REGION Network 29: T-03.00 Transfer Pump Cmd and Speed
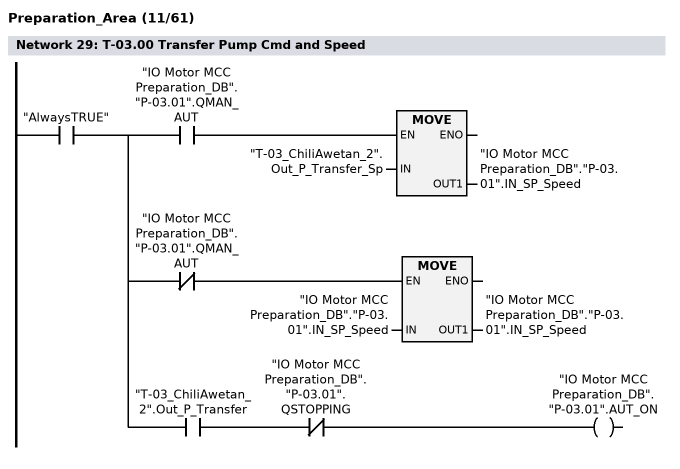
   RUNG wire#powerrail
      Contact( "AlwaysTRUE" )
      wire#w1
      Contact( "IO Motor MCC Preparation_DB"."P-03.01".QMAN_AUT )
      Move(in := "T-03_ChiliAwetan_2".Out_P_Transfer_Sp, out1 => "IO Motor MCC Preparation_DB"."P-03.01".IN_SP_Speed)
   END_RUNG
   RUNG wire#w1
      I_Contact( "IO Motor MCC Preparation_DB"."P-03.01".QMAN_AUT )
      Move(in := "IO Motor MCC Preparation_DB"."P-03.01".IN_SP_Speed, out1 => "IO Motor MCC Preparation_DB"."P-03.01".IN_SP_Speed)
   END_RUNG
   RUNG wire#w1
      Contact( "T-03_ChiliAwetan_2".Out_P_Transfer )
      I_Contact( "IO Motor MCC Preparation_DB"."P-03.01".QSTOPPING )
      Coil( "IO Motor MCC Preparation_DB"."P-03.01".AUT_ON )
   END_RUNG
   // the same network as SCL:
   IF "AlwaysTRUE" AND "IO Motor MCC Preparation_DB"."P-03.01".QMAN_AUT THEN
       "IO Motor MCC Preparation_DB"."P-03.01".IN_SP_Speed := "T-03_ChiliAwetan_2".Out_P_Transfer_Sp;
   END_IF;
   IF "AlwaysTRUE" AND NOT "IO Motor MCC Preparation_DB"."P-03.01".QMAN_AUT THEN
       "IO Motor MCC Preparation_DB"."P-03.01".IN_SP_Speed := "IO Motor MCC Preparation_DB"."P-03.01".IN_SP_Speed;
   END_IF;
   "IO Motor MCC Preparation_DB"."P-03.01".AUT_ON := "AlwaysTRUE" AND "T-03_ChiliAwetan_2".Out_P_Transfer AND NOT "IO Motor MCC Preparation_DB"."P-03.01".QSTOPPING;
END_REGION

REGION Network 30: T-03.00 Feedback Instrument
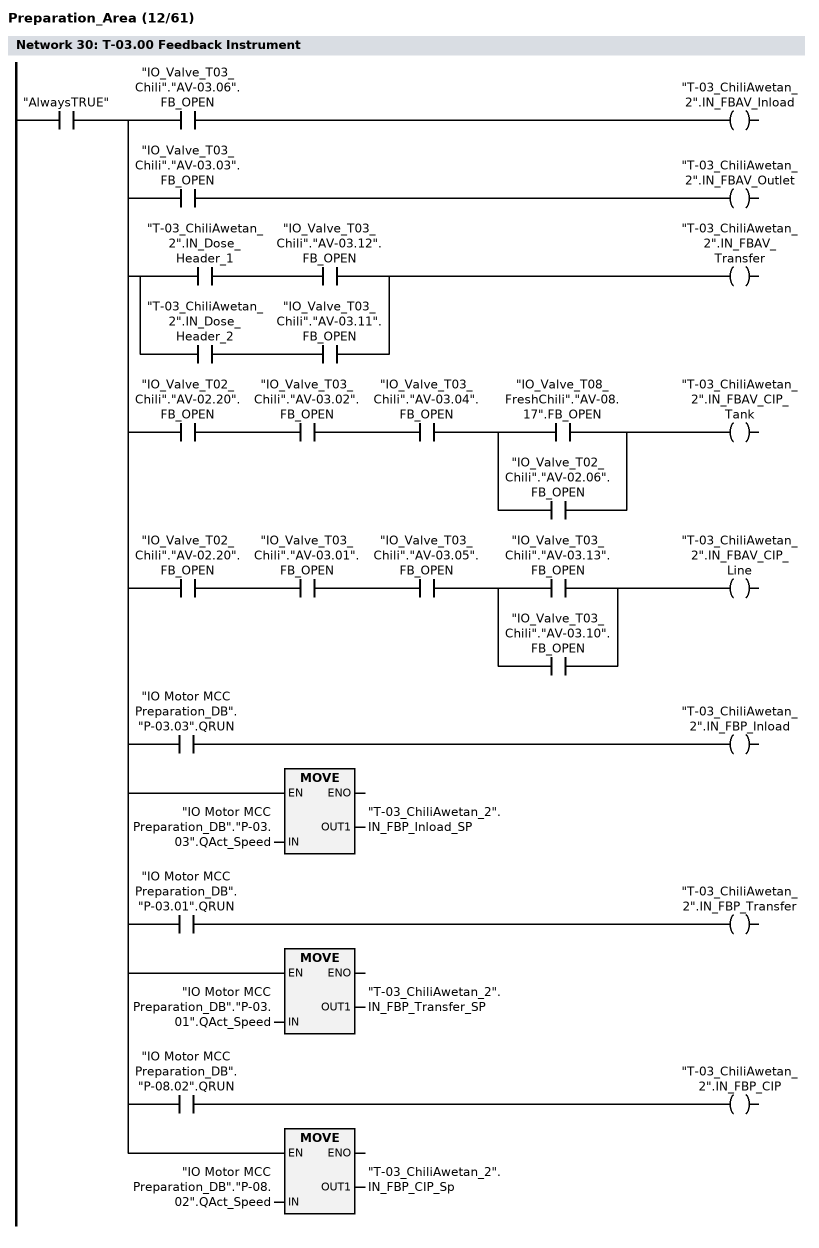
   RUNG wire#powerrail
      Contact( "AlwaysTRUE" )
      wire#w1
      Contact( "IO_Valve_T03_Chili"."AV-03.06".FB_OPEN )
      Coil( "T-03_ChiliAwetan_2".IN_FBAV_Inload )
   END_RUNG
   RUNG wire#w1
      Contact( "IO_Valve_T03_Chili"."AV-03.03".FB_OPEN )
      Coil( "T-03_ChiliAwetan_2".IN_FBAV_Outlet )
   END_RUNG
   RUNG wire#w1
      Contact( "T-03_ChiliAwetan_2".IN_Dose_Header_1 )
      Contact( "IO_Valve_T03_Chili"."AV-03.12".FB_OPEN )
      wire#w2
      Coil( "T-03_ChiliAwetan_2".IN_FBAV_Transfer )
   END_RUNG
   RUNG wire#w1
      Contact( "T-03_ChiliAwetan_2".IN_Dose_Header_2 )
      Contact( "IO_Valve_T03_Chili"."AV-03.11".FB_OPEN )
   END_RUNG wire#w2
   RUNG wire#w1
      Contact( "IO_Valve_T02_Chili"."AV-02.20".FB_OPEN )
      Contact( "IO_Valve_T03_Chili"."AV-03.02".FB_OPEN )
      Contact( "IO_Valve_T03_Chili"."AV-03.04".FB_OPEN )
      wire#w3
      Contact( "IO_Valve_T08_FreshChili"."AV-08.17".FB_OPEN )
      wire#w4
      Coil( "T-03_ChiliAwetan_2".IN_FBAV_CIP_Tank )
   END_RUNG
   RUNG wire#w3
      Contact( "IO_Valve_T02_Chili"."AV-02.06".FB_OPEN )
   END_RUNG wire#w4
   RUNG wire#w1
      Contact( "IO_Valve_T02_Chili"."AV-02.20".FB_OPEN )
      Contact( "IO_Valve_T03_Chili"."AV-03.01".FB_OPEN )
      Contact( "IO_Valve_T03_Chili"."AV-03.05".FB_OPEN )
      wire#w5
      Contact( "IO_Valve_T03_Chili"."AV-03.13".FB_OPEN )
      wire#w6
      Coil( "T-03_ChiliAwetan_2".IN_FBAV_CIP_Line )
   END_RUNG
   RUNG wire#w5
      Contact( "IO_Valve_T03_Chili"."AV-03.10".FB_OPEN )
   END_RUNG wire#w6
   RUNG wire#w1
      Contact( "IO Motor MCC Preparation_DB"."P-03.03".QRUN )
      Coil( "T-03_ChiliAwetan_2".IN_FBP_Inload )
   END_RUNG
   RUNG wire#w1
      Move(in := "IO Motor MCC Preparation_DB"."P-03.03".QAct_Speed, out1 => "T-03_ChiliAwetan_2".IN_FBP_Inload_SP)
   END_RUNG
   RUNG wire#w1
      Contact( "IO Motor MCC Preparation_DB"."P-03.01".QRUN )
      Coil( "T-03_ChiliAwetan_2".IN_FBP_Transfer )
   END_RUNG
   RUNG wire#w1
      Move(in := "IO Motor MCC Preparation_DB"."P-03.01".QAct_Speed, out1 => "T-03_ChiliAwetan_2".IN_FBP_Transfer_SP)
   END_RUNG
   RUNG wire#w1
      Contact( "IO Motor MCC Preparation_DB"."P-08.02".QRUN )
      Coil( "T-03_ChiliAwetan_2".IN_FBP_CIP )
   END_RUNG
   RUNG wire#w1
      Move(in := "IO Motor MCC Preparation_DB"."P-08.02".QAct_Speed, out1 => "T-03_ChiliAwetan_2".IN_FBP_CIP_Sp)
   END_RUNG
   // the same network as SCL:
   "T-03_ChiliAwetan_2".IN_FBAV_Inload := "AlwaysTRUE" AND "IO_Valve_T03_Chili"."AV-03.06".FB_OPEN;
   "T-03_ChiliAwetan_2".IN_FBAV_Outlet := "AlwaysTRUE" AND "IO_Valve_T03_Chili"."AV-03.03".FB_OPEN;
   "T-03_ChiliAwetan_2".IN_FBAV_Transfer := "AlwaysTRUE" AND (("T-03_ChiliAwetan_2".IN_Dose_Header_1 AND "IO_Valve_T03_Chili"."AV-03.12".FB_OPEN) OR ("T-03_ChiliAwetan_2".IN_Dose_Header_2 AND "IO_Valve_T03_Chili"."AV-03.11".FB_OPEN));
   "T-03_ChiliAwetan_2".IN_FBAV_CIP_Tank := "AlwaysTRUE" AND "IO_Valve_T02_Chili"."AV-02.20".FB_OPEN AND "IO_Valve_T03_Chili"."AV-03.02".FB_OPEN AND "IO_Valve_T03_Chili"."AV-03.04".FB_OPEN AND ("IO_Valve_T08_FreshChili"."AV-08.17".FB_OPEN OR "IO_Valve_T02_Chili"."AV-02.06".FB_OPEN);
   "T-03_ChiliAwetan_2".IN_FBAV_CIP_Line := "AlwaysTRUE" AND "IO_Valve_T02_Chili"."AV-02.20".FB_OPEN AND "IO_Valve_T03_Chili"."AV-03.01".FB_OPEN AND "IO_Valve_T03_Chili"."AV-03.05".FB_OPEN AND ("IO_Valve_T03_Chili"."AV-03.13".FB_OPEN OR "IO_Valve_T03_Chili"."AV-03.10".FB_OPEN);
   "T-03_ChiliAwetan_2".IN_FBP_Inload := "AlwaysTRUE" AND "IO Motor MCC Preparation_DB"."P-03.03".QRUN;
   IF "AlwaysTRUE" THEN
       "T-03_ChiliAwetan_2".IN_FBP_Inload_SP := "IO Motor MCC Preparation_DB"."P-03.03".QAct_Speed;
   END_IF;
   "T-03_ChiliAwetan_2".IN_FBP_Transfer := "AlwaysTRUE" AND "IO Motor MCC Preparation_DB"."P-03.01".QRUN;
   IF "AlwaysTRUE" THEN
       "T-03_ChiliAwetan_2".IN_FBP_Transfer_SP := "IO Motor MCC Preparation_DB"."P-03.01".QAct_Speed;
   END_IF;
   "T-03_ChiliAwetan_2".IN_FBP_CIP := "AlwaysTRUE" AND "IO Motor MCC Preparation_DB"."P-08.02".QRUN;
   IF "AlwaysTRUE" THEN
       "T-03_ChiliAwetan_2".IN_FBP_CIP_Sp := "IO Motor MCC Preparation_DB"."P-08.02".QAct_Speed;
   END_IF;
END_REGION

REGION Network 31: T-03.00 Comm to Blend
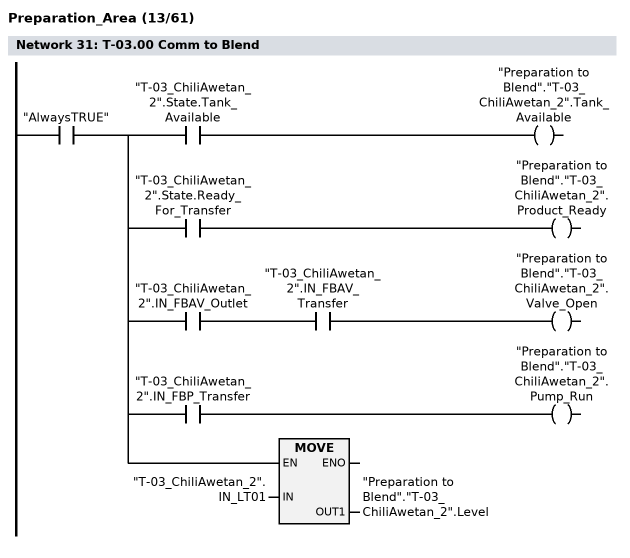
   RUNG wire#powerrail
      Contact( "AlwaysTRUE" )
      wire#w1
      Contact( "T-03_ChiliAwetan_2".State.Tank_Available )
      Coil( "Preparation to Blend"."T-03_ChiliAwetan_2".Tank_Available )
   END_RUNG
   RUNG wire#w1
      Contact( "T-03_ChiliAwetan_2".State.Ready_For_Transfer )
      Coil( "Preparation to Blend"."T-03_ChiliAwetan_2".Product_Ready )
   END_RUNG
   RUNG wire#w1
      Contact( "T-03_ChiliAwetan_2".IN_FBAV_Outlet )
      Contact( "T-03_ChiliAwetan_2".IN_FBAV_Transfer )
      Coil( "Preparation to Blend"."T-03_ChiliAwetan_2".Valve_Open )
   END_RUNG
   RUNG wire#w1
      Contact( "T-03_ChiliAwetan_2".IN_FBP_Transfer )
      Coil( "Preparation to Blend"."T-03_ChiliAwetan_2".Pump_Run )
   END_RUNG
   RUNG wire#w1
      Move(in := "T-03_ChiliAwetan_2".IN_LT01, out1 => "Preparation to Blend"."T-03_ChiliAwetan_2".Level)
   END_RUNG
   // the same network as SCL:
   "Preparation to Blend"."T-03_ChiliAwetan_2".Tank_Available := "AlwaysTRUE" AND "T-03_ChiliAwetan_2".State.Tank_Available;
   "Preparation to Blend"."T-03_ChiliAwetan_2".Product_Ready := "AlwaysTRUE" AND "T-03_ChiliAwetan_2".State.Ready_For_Transfer;
   "Preparation to Blend"."T-03_ChiliAwetan_2".Valve_Open := "AlwaysTRUE" AND "T-03_ChiliAwetan_2".IN_FBAV_Outlet AND "T-03_ChiliAwetan_2".IN_FBAV_Transfer;
   "Preparation to Blend"."T-03_ChiliAwetan_2".Pump_Run := "AlwaysTRUE" AND "T-03_ChiliAwetan_2".IN_FBP_Transfer;
   IF "AlwaysTRUE" THEN
       "Preparation to Blend"."T-03_ChiliAwetan_2".Level := "T-03_ChiliAwetan_2".IN_LT01;
   END_IF;
END_REGION

NETWORK
TITLE = T-04.00 DOSE ON OFF
      O     "Blend to Preparation"."T-20".Raw_Material.ChiliAwetan_3.DoseRun;
      O     "Blend to Preparation"."T-21".Raw_Material.ChiliAwetan_3.DoseRun;
      O     "Blend to Preparation"."T-30".Raw_Material.ChiliAwetan_3.DoseRun;
      O     "Blend to Preparation"."T-31".Raw_Material.ChiliAwetan_3.DoseRun;
      O     "Blend to Preparation"."T-40".Raw_Material.ChiliAwetan_3.DoseRun;
      O     "Blend to Preparation"."T-41".Raw_Material.ChiliAwetan_3.DoseRun;
      =     "T-04_ChiliAwetan_3".IN_Dose_Run;

NETWORK
TITLE = T-04.00 DOSE PAUSE
      O     "Blend to Preparation"."T-20".Raw_Material.ChiliAwetan_3.DoseHeld;
      O     "Blend to Preparation"."T-21".Raw_Material.ChiliAwetan_3.DoseHeld;
      O     "Blend to Preparation"."T-30".Raw_Material.ChiliAwetan_3.DoseHeld;
      O     "Blend to Preparation"."T-31".Raw_Material.ChiliAwetan_3.DoseHeld;
      O     "Blend to Preparation"."T-40".Raw_Material.ChiliAwetan_3.DoseHeld;
      O     "Blend to Preparation"."T-41".Raw_Material.ChiliAwetan_3.DoseHeld;
      =     "T-04_ChiliAwetan_3".IN_Dose_Held;

NETWORK
TITLE = T-04.00 DOSE VALVE CMD
      O(;
      A     "Blend to Preparation"."T-20".Raw_Material.ChiliAwetan_3.DoseRun;
      A     "Blend to Preparation"."T-20".Raw_Material.ChiliAwetan_3.ValveCMD;
      );
      O(;
      A     "Blend to Preparation"."T-21".Raw_Material.ChiliAwetan_3.DoseRun;
      A     "Blend to Preparation"."T-21".Raw_Material.ChiliAwetan_3.ValveCMD;
      );
      O(;
      A     "Blend to Preparation"."T-30".Raw_Material.ChiliAwetan_3.DoseRun;
      A     "Blend to Preparation"."T-30".Raw_Material.ChiliAwetan_3.ValveCMD;
      );
      O(;
      A     "Blend to Preparation"."T-31".Raw_Material.ChiliAwetan_3.DoseRun;
      A     "Blend to Preparation"."T-31".Raw_Material.ChiliAwetan_3.ValveCMD;
      );
      O(;
      A     "Blend to Preparation"."T-40".Raw_Material.ChiliAwetan_3.DoseRun;
      A     "Blend to Preparation"."T-40".Raw_Material.ChiliAwetan_3.ValveCMD;
      );
      O(;
      A     "Blend to Preparation"."T-41".Raw_Material.ChiliAwetan_3.DoseRun;
      A     "Blend to Preparation"."T-41".Raw_Material.ChiliAwetan_3.ValveCMD;
      );
      =     "T-04_ChiliAwetan_3".IN_Dose_Valve_Cmd;



NETWORK
TITLE = T-04.00 DOSE Pump CMD
      O(;
      A     "Blend to Preparation"."T-20".Raw_Material.ChiliAwetan_3.DoseRun;
      A     "Blend to Preparation"."T-20".Raw_Material.ChiliAwetan_3.PumpCMD;
      );
      O(;
      A     "Blend to Preparation"."T-21".Raw_Material.ChiliAwetan_3.DoseRun;
      A     "Blend to Preparation"."T-21".Raw_Material.ChiliAwetan_3.PumpCMD;
      );
      O(;
      A     "Blend to Preparation"."T-30".Raw_Material.ChiliAwetan_3.DoseRun;
      A     "Blend to Preparation"."T-30".Raw_Material.ChiliAwetan_3.PumpCMD;
      );
      O(;
      A     "Blend to Preparation"."T-31".Raw_Material.ChiliAwetan_3.DoseRun;
      A     "Blend to Preparation"."T-31".Raw_Material.ChiliAwetan_3.PumpCMD;
      );
      O(;
      A     "Blend to Preparation"."T-40".Raw_Material.ChiliAwetan_3.DoseRun;
      A     "Blend to Preparation"."T-40".Raw_Material.ChiliAwetan_3.PumpCMD;
      );
      O(;
      A     "Blend to Preparation"."T-41".Raw_Material.ChiliAwetan_3.DoseRun;
      A     "Blend to Preparation"."T-41".Raw_Material.ChiliAwetan_3.PumpCMD;
      );
      =     "T-04_ChiliAwetan_3".IN_Dose_Pump_Cmd;



NETWORK
TITLE = T-04.00 DOSE PUMP SPEED
// Checking
      O     "Blend to Preparation"."T-20".Raw_Material.ChiliAwetan_3.DoseRun;
      JC    SP_04_FROM_20;
      O     "Blend to Preparation"."T-21".Raw_Material.ChiliAwetan_3.DoseRun;
      JC    SP_04_FROM_21;
      O     "Blend to Preparation"."T-30".Raw_Material.ChiliAwetan_3.DoseRun;
      JC    SP_04_FROM_30;
      O     "Blend to Preparation"."T-31".Raw_Material.ChiliAwetan_3.DoseRun;
      JC    SP_04_FROM_31;
      O     "Blend to Preparation"."T-40".Raw_Material.ChiliAwetan_3.DoseRun;
      JC    SP_04_FROM_40;
      O     "Blend to Preparation"."T-41".Raw_Material.ChiliAwetan_3.DoseRun;
      JC    SP_04_FROM_41;
//Jump to end if Blend not Dosing
      JC    SP_04_SELF;
//Load Set Point
SP_04_FROM_20:L     "Blend to Preparation".Recipe."T-20".ChiliAwetan_3.SP_PumpSpeed;
      T     "T-04_ChiliAwetan_3".IN_Dose_Pump_Sp;
      JC    SP_04_SELF;
SP_04_FROM_21:L     "Blend to Preparation".Recipe."T-21".ChiliAwetan_3.SP_PumpSpeed;
      T     "T-04_ChiliAwetan_3".IN_Dose_Pump_Sp;
      JC    SP_04_SELF;
SP_04_FROM_30:L     "Blend to Preparation".Recipe."T-30".ChiliAwetan_3.SP_PumpSpeed;
      T     "T-04_ChiliAwetan_3".IN_Dose_Pump_Sp;
      JC    SP_04_SELF;
SP_04_FROM_31:L     "Blend to Preparation".Recipe."T-31".ChiliAwetan_3.SP_PumpSpeed;
      T     "T-04_ChiliAwetan_3".IN_Dose_Pump_Sp;
      JC    SP_04_SELF;
SP_04_FROM_40:L     "Blend to Preparation".Recipe."T-40".ChiliAwetan_3.SP_PumpSpeed;
      T     "T-04_ChiliAwetan_3".IN_Dose_Pump_Sp;
      JC    SP_04_SELF;
SP_04_FROM_41:L     "Blend to Preparation".Recipe."T-41".ChiliAwetan_3.SP_PumpSpeed;
      T     "T-04_ChiliAwetan_3".IN_Dose_Pump_Sp;
      JC    SP_04_SELF;
// END
SP_04_SELF:L     "T-04_ChiliAwetan_3".IN_Dose_Pump_Sp;
      T     "T-04_ChiliAwetan_3".IN_Dose_Pump_Sp;


NETWORK
TITLE = T-04.00 Header Req
// HEADER 1 Req
      O     "Blend to Preparation"."T-20".Raw_Material.ChiliAwetan_3.Header1_Req;
      O     "Blend to Preparation"."T-21".Raw_Material.ChiliAwetan_3.Header1_Req;
      O     "Blend to Preparation"."T-30".Raw_Material.ChiliAwetan_3.Header1_Req;
      O     "Blend to Preparation"."T-31".Raw_Material.ChiliAwetan_3.Header1_Req;
      O     "Blend to Preparation"."T-40".Raw_Material.ChiliAwetan_3.Header1_Req;
      O     "Blend to Preparation"."T-41".Raw_Material.ChiliAwetan_3.Header1_Req;
      =     "T-04_ChiliAwetan_3".IN_Dose_Header_1;

// HEADER 2 Req
      O     "Blend to Preparation"."T-20".Raw_Material.ChiliAwetan_3.Header2_Req;
      O     "Blend to Preparation"."T-21".Raw_Material.ChiliAwetan_3.Header2_Req;
      O     "Blend to Preparation"."T-30".Raw_Material.ChiliAwetan_3.Header2_Req;
      O     "Blend to Preparation"."T-31".Raw_Material.ChiliAwetan_3.Header2_Req;
      O     "Blend to Preparation"."T-40".Raw_Material.ChiliAwetan_3.Header2_Req;
      O     "Blend to Preparation"."T-41".Raw_Material.ChiliAwetan_3.Header2_Req;
      =     "T-04_ChiliAwetan_3".IN_Dose_Header_2;


REGION Network 40: T-04.00 LineTransferOK
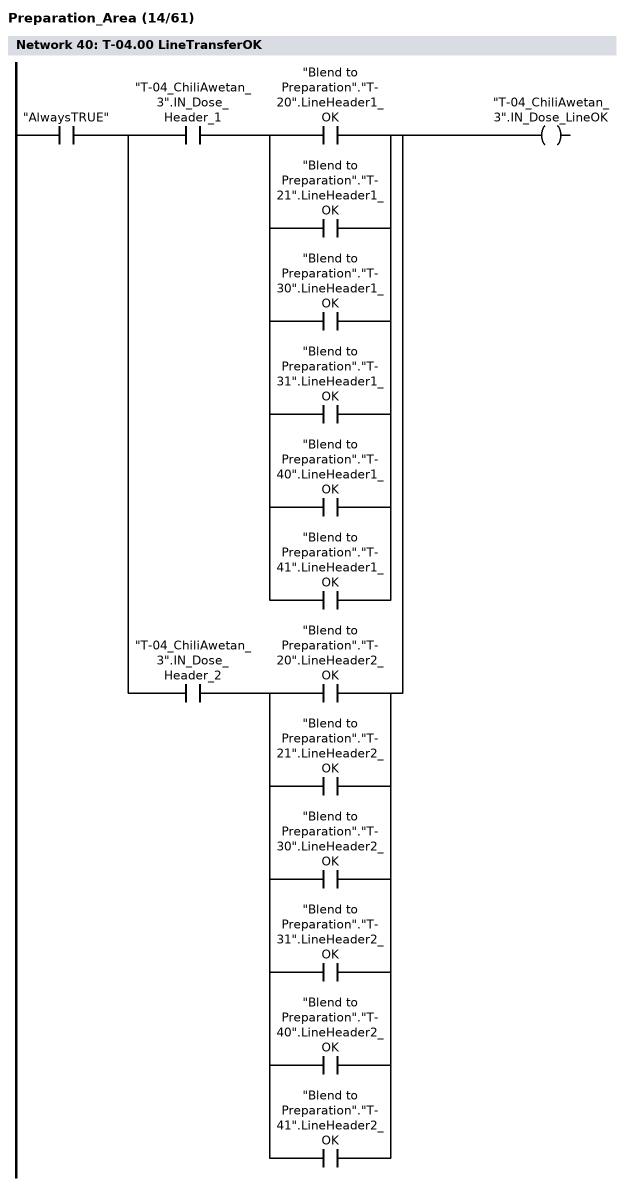
   RUNG wire#powerrail
      Contact( "AlwaysTRUE" )
      wire#w1
      Contact( "T-04_ChiliAwetan_3".IN_Dose_Header_1 )
      wire#w2
      Contact( "Blend to Preparation"."T-20".LineHeader1_OK )
      wire#w3
      Coil( "T-04_ChiliAwetan_3".IN_Dose_LineOK )
   END_RUNG
   RUNG wire#w2
      Contact( "Blend to Preparation"."T-21".LineHeader1_OK )
   END_RUNG wire#w3
   RUNG wire#w2
      Contact( "Blend to Preparation"."T-30".LineHeader1_OK )
   END_RUNG wire#w3
   RUNG wire#w2
      Contact( "Blend to Preparation"."T-31".LineHeader1_OK )
   END_RUNG wire#w3
   RUNG wire#w2
      Contact( "Blend to Preparation"."T-40".LineHeader1_OK )
   END_RUNG wire#w3
   RUNG wire#w2
      Contact( "Blend to Preparation"."T-41".LineHeader1_OK )
   END_RUNG wire#w3
   RUNG wire#w1
      Contact( "T-04_ChiliAwetan_3".IN_Dose_Header_2 )
      wire#w4
      Contact( "Blend to Preparation"."T-20".LineHeader2_OK )
   END_RUNG wire#w3
   RUNG wire#w4
      Contact( "Blend to Preparation"."T-21".LineHeader2_OK )
   END_RUNG wire#w3
   RUNG wire#w4
      Contact( "Blend to Preparation"."T-30".LineHeader2_OK )
   END_RUNG wire#w3
   RUNG wire#w4
      Contact( "Blend to Preparation"."T-31".LineHeader2_OK )
   END_RUNG wire#w3
   RUNG wire#w4
      Contact( "Blend to Preparation"."T-40".LineHeader2_OK )
   END_RUNG wire#w3
   RUNG wire#w4
      Contact( "Blend to Preparation"."T-41".LineHeader2_OK )
   END_RUNG wire#w3
   // the same network as SCL:
   "T-04_ChiliAwetan_3".IN_Dose_LineOK := "AlwaysTRUE" AND (("T-04_ChiliAwetan_3".IN_Dose_Header_1 AND ("Blend to Preparation"."T-20".LineHeader1_OK OR "Blend to Preparation"."T-21".LineHeader1_OK OR "Blend to Preparation"."T-30".LineHeader1_OK OR "Blend to Preparation"."T-31".LineHeader1_OK OR "Blend to Preparation"."T-40".LineHeader1_OK OR "Blend to Preparation"."T-41".LineHeader1_OK)) OR ("T-04_ChiliAwetan_3".IN_Dose_Header_2 AND ("Blend to Preparation"."T-20".LineHeader2_OK OR "Blend to Preparation"."T-21".LineHeader2_OK OR "Blend to Preparation"."T-30".LineHeader2_OK OR "Blend to Preparation"."T-31".LineHeader2_OK OR "Blend to Preparation"."T-40".LineHeader2_OK OR "Blend to Preparation"."T-41".LineHeader2_OK)));
END_REGION

REGION Network 41: T-04.00___Chili Awetan 3
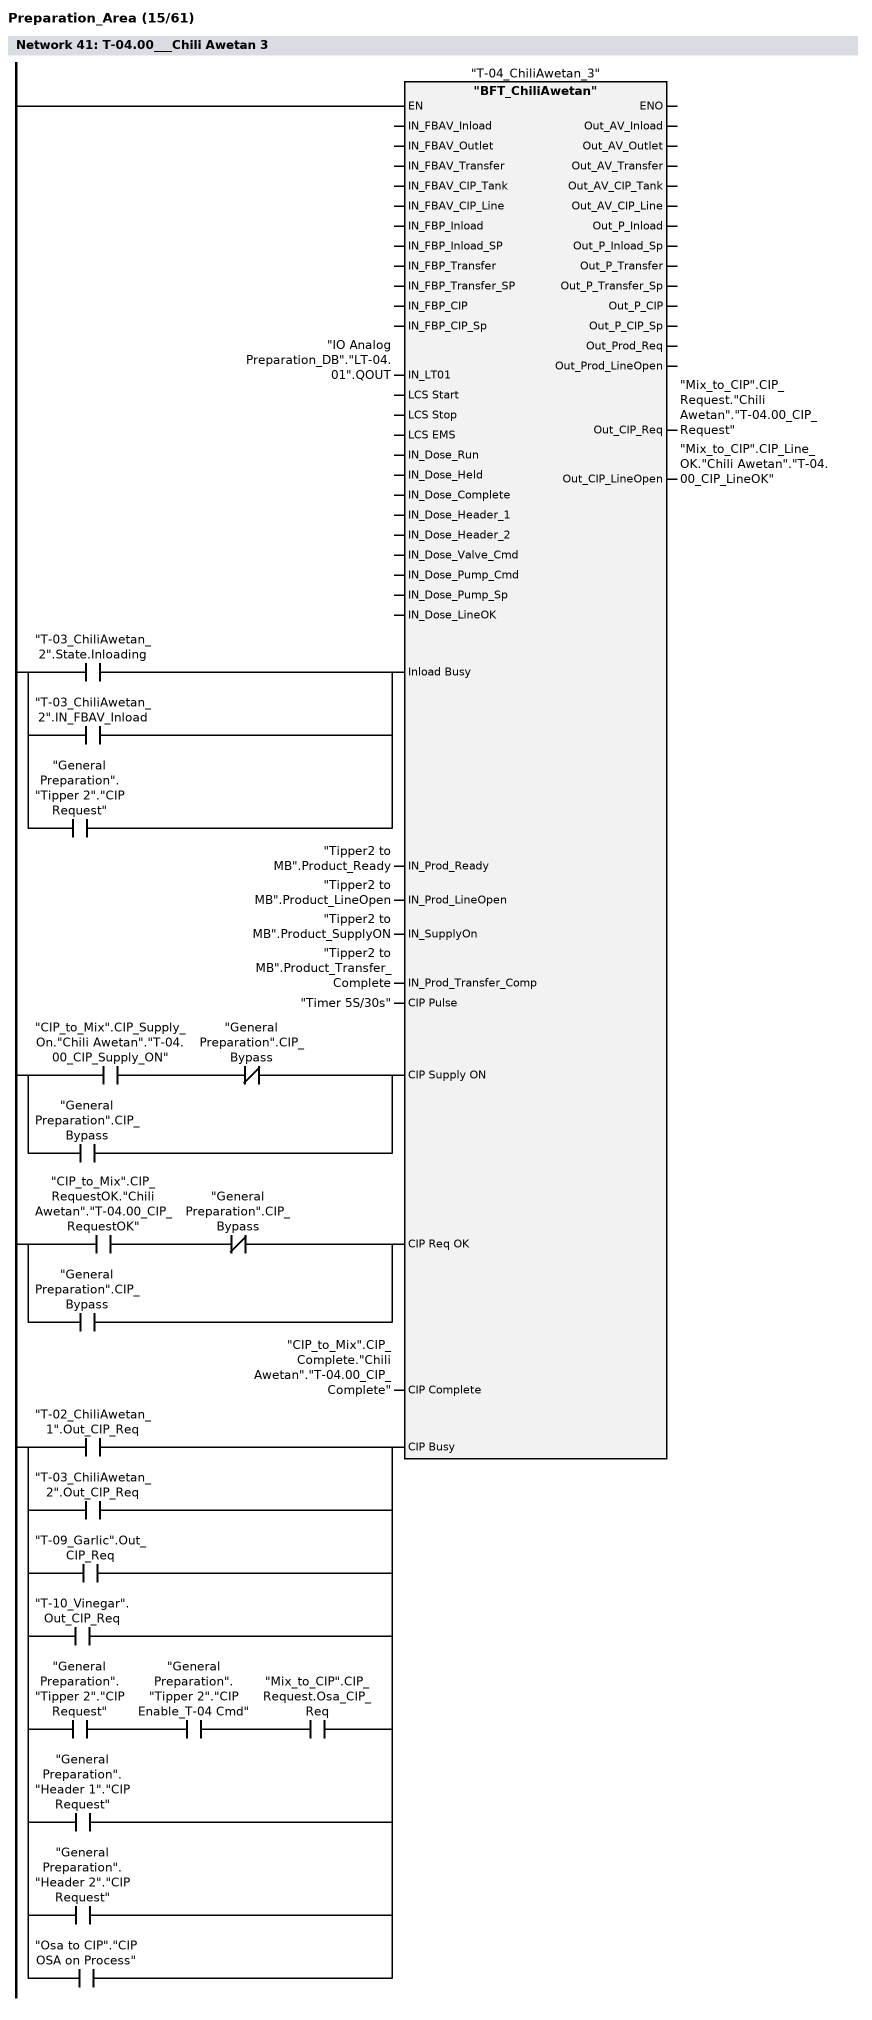
   RUNG wire#powerrail
      "T-04_ChiliAwetan_3"("Inload Busy" := wire#w1, "CIP Supply ON" := wire#w2, "CIP Req OK" := wire#w3, "CIP Busy" := wire#w4, IN_FBAV_Inload :=, IN_FBAV_Outlet :=, IN_FBAV_Transfer :=, IN_FBAV_CIP_Tank :=, IN_FBAV_CIP_Line :=, IN_FBP_Inload :=, IN_FBP_Inload_SP :=, IN_FBP_Transfer :=, IN_FBP_Transfer_SP :=, IN_FBP_CIP :=, IN_FBP_CIP_Sp :=, IN_LT01 := "IO Analog Preparation_DB"."LT-04.01".QOUT, "LCS Start" :=, "LCS Stop" :=, "LCS EMS" :=, IN_Dose_Run :=, IN_Dose_Held :=, IN_Dose_Complete :=, IN_Dose_Header_1 :=, IN_Dose_Header_2 :=, IN_Dose_Valve_Cmd :=, IN_Dose_Pump_Cmd :=, IN_Dose_Pump_Sp :=, IN_Dose_LineOK :=, IN_Prod_Ready := "Tipper2 to MB".Product_Ready, IN_Prod_LineOpen := "Tipper2 to MB".Product_LineOpen, IN_SupplyOn := "Tipper2 to MB".Product_SupplyON, IN_Prod_Transfer_Comp := "Tipper2 to MB".Product_Transfer_Complete, "CIP Pulse" := "Timer 5S/30s", "CIP Complete" := "CIP_to_Mix".CIP_Complete."Chili Awetan"."T-04.00_CIP_Complete", Out_AV_Inload =>, Out_AV_Outlet =>, Out_AV_Transfer =>, Out_AV_CIP_Tank =>, Out_AV_CIP_Line =>, Out_P_Inload =>, Out_P_Inload_Sp =>, Out_P_Transfer =>, Out_P_Transfer_Sp =>, Out_P_CIP =>, Out_P_CIP_Sp =>, Out_Prod_Req =>, Out_Prod_LineOpen =>, Out_CIP_Req => "Mix_to_CIP".CIP_Request."Chili Awetan"."T-04.00_CIP_Request", Out_CIP_LineOpen => "Mix_to_CIP".CIP_Line_OK."Chili Awetan"."T-04.00_CIP_LineOK")
   END_RUNG
   RUNG wire#powerrail
      Contact( "T-03_ChiliAwetan_2".State.Inloading )
   END_RUNG wire#w1
   RUNG wire#powerrail
      Contact( "T-03_ChiliAwetan_2".IN_FBAV_Inload )
   END_RUNG wire#w1
   RUNG wire#powerrail
      Contact( "General Preparation"."Tipper 2"."CIP Request" )
   END_RUNG wire#w1
   RUNG wire#powerrail
      Contact( "CIP_to_Mix".CIP_Supply_On."Chili Awetan"."T-04.00_CIP_Supply_ON" )
      I_Contact( "General Preparation".CIP_Bypass )
   END_RUNG wire#w2
   RUNG wire#powerrail
      Contact( "General Preparation".CIP_Bypass )
   END_RUNG wire#w2
   RUNG wire#powerrail
      Contact( "CIP_to_Mix".CIP_RequestOK."Chili Awetan"."T-04.00_CIP_RequestOK" )
      I_Contact( "General Preparation".CIP_Bypass )
   END_RUNG wire#w3
   RUNG wire#powerrail
      Contact( "General Preparation".CIP_Bypass )
   END_RUNG wire#w3
   RUNG wire#powerrail
      Contact( "T-02_ChiliAwetan_1".Out_CIP_Req )
   END_RUNG wire#w4
   RUNG wire#powerrail
      Contact( "T-03_ChiliAwetan_2".Out_CIP_Req )
   END_RUNG wire#w4
   RUNG wire#powerrail
      Contact( "T-09_Garlic".Out_CIP_Req )
   END_RUNG wire#w4
   RUNG wire#powerrail
      Contact( "T-10_Vinegar".Out_CIP_Req )
   END_RUNG wire#w4
   RUNG wire#powerrail
      Contact( "General Preparation"."Tipper 2"."CIP Request" )
      Contact( "General Preparation"."Tipper 2"."CIP Enable_T-04 Cmd" )
      Contact( "Mix_to_CIP".CIP_Request.Osa_CIP_Req )
   END_RUNG wire#w4
   RUNG wire#powerrail
      Contact( "General Preparation"."Header 1"."CIP Request" )
   END_RUNG wire#w4
   RUNG wire#powerrail
      Contact( "General Preparation"."Header 2"."CIP Request" )
   END_RUNG wire#w4
   RUNG wire#powerrail
      Contact( "Osa to CIP"."CIP OSA on Process" )
   END_RUNG wire#w4
   // the same network as SCL:
   "T-04_ChiliAwetan_3"(IN_LT01 := "IO Analog Preparation_DB"."LT-04.01".QOUT,   // "BFT_ChiliAwetan"
                        "Inload Busy" := "T-03_ChiliAwetan_2".State.Inloading OR "T-03_ChiliAwetan_2".IN_FBAV_Inload OR "General Preparation"."Tipper 2"."CIP Request",
                        IN_Prod_Ready := "Tipper2 to MB".Product_Ready,
                        IN_Prod_LineOpen := "Tipper2 to MB".Product_LineOpen,
                        IN_SupplyOn := "Tipper2 to MB".Product_SupplyON,
                        IN_Prod_Transfer_Comp := "Tipper2 to MB".Product_Transfer_Complete,
                        "CIP Pulse" := "Timer 5S/30s",
                        "CIP Supply ON" := ("CIP_to_Mix".CIP_Supply_On."Chili Awetan"."T-04.00_CIP_Supply_ON" AND NOT "General Preparation".CIP_Bypass) OR "General Preparation".CIP_Bypass,
                        "CIP Req OK" := ("CIP_to_Mix".CIP_RequestOK."Chili Awetan"."T-04.00_CIP_RequestOK" AND NOT "General Preparation".CIP_Bypass) OR "General Preparation".CIP_Bypass,
                        "CIP Complete" := "CIP_to_Mix".CIP_Complete."Chili Awetan"."T-04.00_CIP_Complete",
                        "CIP Busy" := "T-02_ChiliAwetan_1".Out_CIP_Req OR "T-03_ChiliAwetan_2".Out_CIP_Req OR "T-09_Garlic".Out_CIP_Req OR "T-10_Vinegar".Out_CIP_Req OR ("General Preparation"."Tipper 2"."CIP Request" AND "General Preparation"."Tipper 2"."CIP Enable_T-04 Cmd" AND "Mix_to_CIP".CIP_Request.Osa_CIP_Req) OR "General Preparation"."Header 1"."CIP Request" OR "General Preparation"."Header 2"."CIP Request" OR "Osa to CIP"."CIP OSA on Process",
                        Out_CIP_Req => "Mix_to_CIP".CIP_Request."Chili Awetan"."T-04.00_CIP_Request",
                        Out_CIP_LineOpen => "Mix_to_CIP".CIP_Line_OK."Chili Awetan"."T-04.00_CIP_LineOK");
END_REGION

REGION Network 42: T-04.00 Valve Cmd
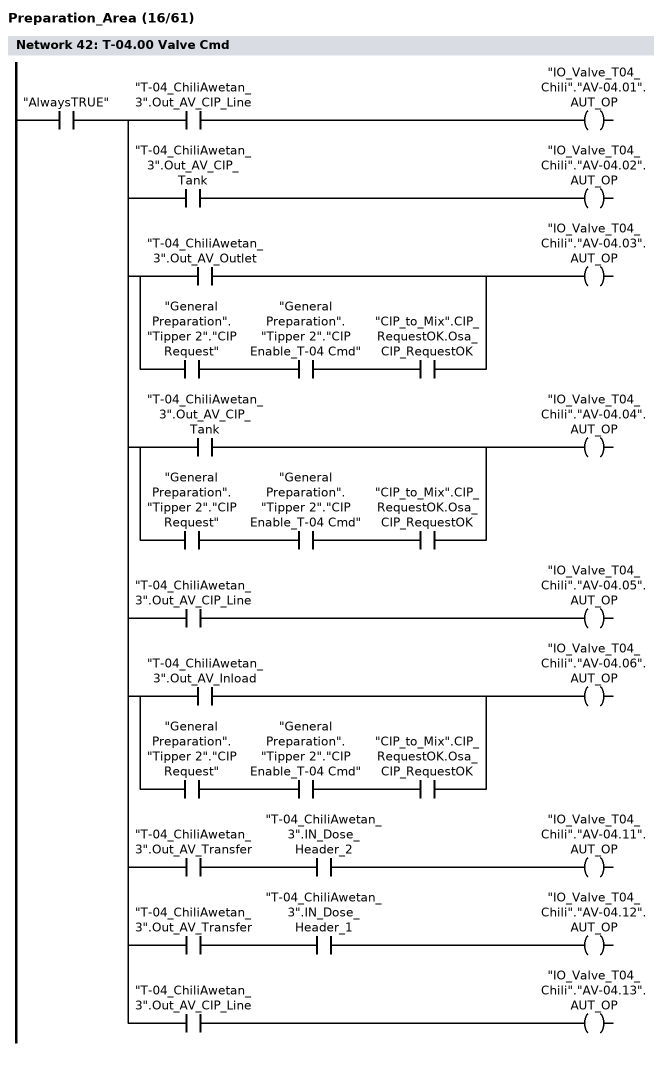
   RUNG wire#powerrail
      Contact( "AlwaysTRUE" )
      wire#w1
      Contact( "T-04_ChiliAwetan_3".Out_AV_CIP_Line )
      Coil( "IO_Valve_T04_Chili"."AV-04.01".AUT_OP )
   END_RUNG
   RUNG wire#w1
      Contact( "T-04_ChiliAwetan_3".Out_AV_CIP_Tank )
      Coil( "IO_Valve_T04_Chili"."AV-04.02".AUT_OP )
   END_RUNG
   RUNG wire#w1
      Contact( "T-04_ChiliAwetan_3".Out_AV_Outlet )
      wire#w2
      Coil( "IO_Valve_T04_Chili"."AV-04.03".AUT_OP )
   END_RUNG
   RUNG wire#w1
      Contact( "General Preparation"."Tipper 2"."CIP Request" )
      Contact( "General Preparation"."Tipper 2"."CIP Enable_T-04 Cmd" )
      Contact( "CIP_to_Mix".CIP_RequestOK.Osa_CIP_RequestOK )
   END_RUNG wire#w2
   RUNG wire#w1
      Contact( "T-04_ChiliAwetan_3".Out_AV_CIP_Tank )
      wire#w3
      Coil( "IO_Valve_T04_Chili"."AV-04.04".AUT_OP )
   END_RUNG
   RUNG wire#w1
      Contact( "General Preparation"."Tipper 2"."CIP Request" )
      Contact( "General Preparation"."Tipper 2"."CIP Enable_T-04 Cmd" )
      Contact( "CIP_to_Mix".CIP_RequestOK.Osa_CIP_RequestOK )
   END_RUNG wire#w3
   RUNG wire#w1
      Contact( "T-04_ChiliAwetan_3".Out_AV_CIP_Line )
      Coil( "IO_Valve_T04_Chili"."AV-04.05".AUT_OP )
   END_RUNG
   RUNG wire#w1
      Contact( "T-04_ChiliAwetan_3".Out_AV_Inload )
      wire#w4
      Coil( "IO_Valve_T04_Chili"."AV-04.06".AUT_OP )
   END_RUNG
   RUNG wire#w1
      Contact( "General Preparation"."Tipper 2"."CIP Request" )
      Contact( "General Preparation"."Tipper 2"."CIP Enable_T-04 Cmd" )
      Contact( "CIP_to_Mix".CIP_RequestOK.Osa_CIP_RequestOK )
   END_RUNG wire#w4
   RUNG wire#w1
      Contact( "T-04_ChiliAwetan_3".Out_AV_Transfer )
      Contact( "T-04_ChiliAwetan_3".IN_Dose_Header_2 )
      Coil( "IO_Valve_T04_Chili"."AV-04.11".AUT_OP )
   END_RUNG
   RUNG wire#w1
      Contact( "T-04_ChiliAwetan_3".Out_AV_Transfer )
      Contact( "T-04_ChiliAwetan_3".IN_Dose_Header_1 )
      Coil( "IO_Valve_T04_Chili"."AV-04.12".AUT_OP )
   END_RUNG
   RUNG wire#w1
      Contact( "T-04_ChiliAwetan_3".Out_AV_CIP_Line )
      Coil( "IO_Valve_T04_Chili"."AV-04.13".AUT_OP )
   END_RUNG
   // the same network as SCL:
   "IO_Valve_T04_Chili"."AV-04.01".AUT_OP := "AlwaysTRUE" AND "T-04_ChiliAwetan_3".Out_AV_CIP_Line;
   "IO_Valve_T04_Chili"."AV-04.02".AUT_OP := "AlwaysTRUE" AND "T-04_ChiliAwetan_3".Out_AV_CIP_Tank;
   "IO_Valve_T04_Chili"."AV-04.03".AUT_OP := "AlwaysTRUE" AND ("T-04_ChiliAwetan_3".Out_AV_Outlet OR ("General Preparation"."Tipper 2"."CIP Request" AND "General Preparation"."Tipper 2"."CIP Enable_T-04 Cmd" AND "CIP_to_Mix".CIP_RequestOK.Osa_CIP_RequestOK));
   "IO_Valve_T04_Chili"."AV-04.04".AUT_OP := "AlwaysTRUE" AND ("T-04_ChiliAwetan_3".Out_AV_CIP_Tank OR ("General Preparation"."Tipper 2"."CIP Request" AND "General Preparation"."Tipper 2"."CIP Enable_T-04 Cmd" AND "CIP_to_Mix".CIP_RequestOK.Osa_CIP_RequestOK));
   "IO_Valve_T04_Chili"."AV-04.05".AUT_OP := "AlwaysTRUE" AND "T-04_ChiliAwetan_3".Out_AV_CIP_Line;
   "IO_Valve_T04_Chili"."AV-04.06".AUT_OP := "AlwaysTRUE" AND ("T-04_ChiliAwetan_3".Out_AV_Inload OR ("General Preparation"."Tipper 2"."CIP Request" AND "General Preparation"."Tipper 2"."CIP Enable_T-04 Cmd" AND "CIP_to_Mix".CIP_RequestOK.Osa_CIP_RequestOK));
   "IO_Valve_T04_Chili"."AV-04.11".AUT_OP := "AlwaysTRUE" AND "T-04_ChiliAwetan_3".Out_AV_Transfer AND "T-04_ChiliAwetan_3".IN_Dose_Header_2;
   "IO_Valve_T04_Chili"."AV-04.12".AUT_OP := "AlwaysTRUE" AND "T-04_ChiliAwetan_3".Out_AV_Transfer AND "T-04_ChiliAwetan_3".IN_Dose_Header_1;
   "IO_Valve_T04_Chili"."AV-04.13".AUT_OP := "AlwaysTRUE" AND "T-04_ChiliAwetan_3".Out_AV_CIP_Line;
END_REGION

REGION Network 43: T-04.00 Transfer Pump Cmd and Speed
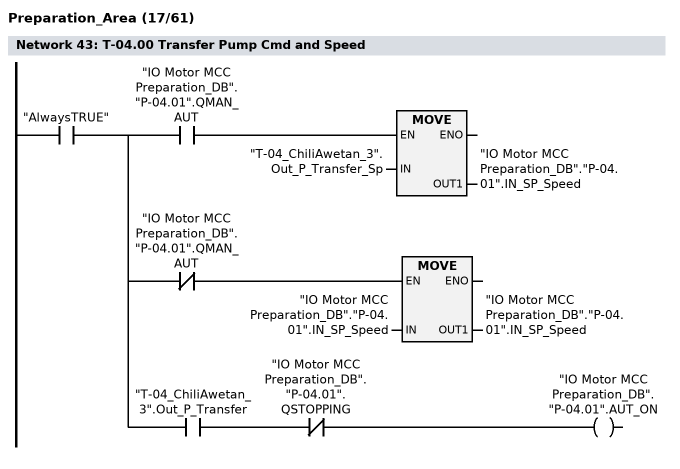
   RUNG wire#powerrail
      Contact( "AlwaysTRUE" )
      wire#w1
      Contact( "IO Motor MCC Preparation_DB"."P-04.01".QMAN_AUT )
      Move(in := "T-04_ChiliAwetan_3".Out_P_Transfer_Sp, out1 => "IO Motor MCC Preparation_DB"."P-04.01".IN_SP_Speed)
   END_RUNG
   RUNG wire#w1
      I_Contact( "IO Motor MCC Preparation_DB"."P-04.01".QMAN_AUT )
      Move(in := "IO Motor MCC Preparation_DB"."P-04.01".IN_SP_Speed, out1 => "IO Motor MCC Preparation_DB"."P-04.01".IN_SP_Speed)
   END_RUNG
   RUNG wire#w1
      Contact( "T-04_ChiliAwetan_3".Out_P_Transfer )
      I_Contact( "IO Motor MCC Preparation_DB"."P-04.01".QSTOPPING )
      Coil( "IO Motor MCC Preparation_DB"."P-04.01".AUT_ON )
   END_RUNG
   // the same network as SCL:
   IF "AlwaysTRUE" AND "IO Motor MCC Preparation_DB"."P-04.01".QMAN_AUT THEN
       "IO Motor MCC Preparation_DB"."P-04.01".IN_SP_Speed := "T-04_ChiliAwetan_3".Out_P_Transfer_Sp;
   END_IF;
   IF "AlwaysTRUE" AND NOT "IO Motor MCC Preparation_DB"."P-04.01".QMAN_AUT THEN
       "IO Motor MCC Preparation_DB"."P-04.01".IN_SP_Speed := "IO Motor MCC Preparation_DB"."P-04.01".IN_SP_Speed;
   END_IF;
   "IO Motor MCC Preparation_DB"."P-04.01".AUT_ON := "AlwaysTRUE" AND "T-04_ChiliAwetan_3".Out_P_Transfer AND NOT "IO Motor MCC Preparation_DB"."P-04.01".QSTOPPING;
END_REGION

REGION Network 44: T-04.00 Feedback Instrument
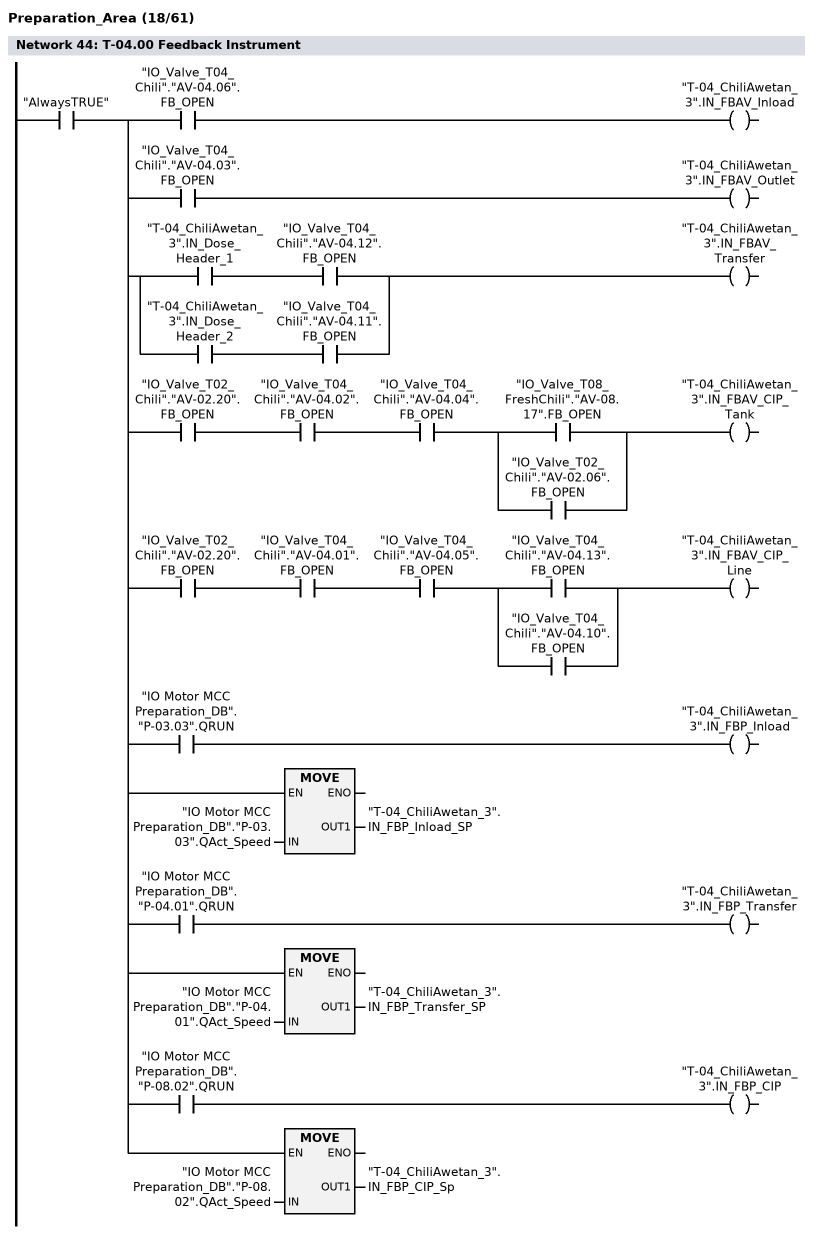
   RUNG wire#powerrail
      Contact( "AlwaysTRUE" )
      wire#w1
      Contact( "IO_Valve_T04_Chili"."AV-04.06".FB_OPEN )
      Coil( "T-04_ChiliAwetan_3".IN_FBAV_Inload )
   END_RUNG
   RUNG wire#w1
      Contact( "IO_Valve_T04_Chili"."AV-04.03".FB_OPEN )
      Coil( "T-04_ChiliAwetan_3".IN_FBAV_Outlet )
   END_RUNG
   RUNG wire#w1
      Contact( "T-04_ChiliAwetan_3".IN_Dose_Header_1 )
      Contact( "IO_Valve_T04_Chili"."AV-04.12".FB_OPEN )
      wire#w2
      Coil( "T-04_ChiliAwetan_3".IN_FBAV_Transfer )
   END_RUNG
   RUNG wire#w1
      Contact( "T-04_ChiliAwetan_3".IN_Dose_Header_2 )
      Contact( "IO_Valve_T04_Chili"."AV-04.11".FB_OPEN )
   END_RUNG wire#w2
   RUNG wire#w1
      Contact( "IO_Valve_T02_Chili"."AV-02.20".FB_OPEN )
      Contact( "IO_Valve_T04_Chili"."AV-04.02".FB_OPEN )
      Contact( "IO_Valve_T04_Chili"."AV-04.04".FB_OPEN )
      wire#w3
      Contact( "IO_Valve_T08_FreshChili"."AV-08.17".FB_OPEN )
      wire#w4
      Coil( "T-04_ChiliAwetan_3".IN_FBAV_CIP_Tank )
   END_RUNG
   RUNG wire#w3
      Contact( "IO_Valve_T02_Chili"."AV-02.06".FB_OPEN )
   END_RUNG wire#w4
   RUNG wire#w1
      Contact( "IO_Valve_T02_Chili"."AV-02.20".FB_OPEN )
      Contact( "IO_Valve_T04_Chili"."AV-04.01".FB_OPEN )
      Contact( "IO_Valve_T04_Chili"."AV-04.05".FB_OPEN )
      wire#w5
      Contact( "IO_Valve_T04_Chili"."AV-04.13".FB_OPEN )
      wire#w6
      Coil( "T-04_ChiliAwetan_3".IN_FBAV_CIP_Line )
   END_RUNG
   RUNG wire#w5
      Contact( "IO_Valve_T04_Chili"."AV-04.10".FB_OPEN )
   END_RUNG wire#w6
   RUNG wire#w1
      Contact( "IO Motor MCC Preparation_DB"."P-03.03".QRUN )
      Coil( "T-04_ChiliAwetan_3".IN_FBP_Inload )
   END_RUNG
   RUNG wire#w1
      Move(in := "IO Motor MCC Preparation_DB"."P-03.03".QAct_Speed, out1 => "T-04_ChiliAwetan_3".IN_FBP_Inload_SP)
   END_RUNG
   RUNG wire#w1
      Contact( "IO Motor MCC Preparation_DB"."P-04.01".QRUN )
      Coil( "T-04_ChiliAwetan_3".IN_FBP_Transfer )
   END_RUNG
   RUNG wire#w1
      Move(in := "IO Motor MCC Preparation_DB"."P-04.01".QAct_Speed, out1 => "T-04_ChiliAwetan_3".IN_FBP_Transfer_SP)
   END_RUNG
   RUNG wire#w1
      Contact( "IO Motor MCC Preparation_DB"."P-08.02".QRUN )
      Coil( "T-04_ChiliAwetan_3".IN_FBP_CIP )
   END_RUNG
   RUNG wire#w1
      Move(in := "IO Motor MCC Preparation_DB"."P-08.02".QAct_Speed, out1 => "T-04_ChiliAwetan_3".IN_FBP_CIP_Sp)
   END_RUNG
   // the same network as SCL:
   "T-04_ChiliAwetan_3".IN_FBAV_Inload := "AlwaysTRUE" AND "IO_Valve_T04_Chili"."AV-04.06".FB_OPEN;
   "T-04_ChiliAwetan_3".IN_FBAV_Outlet := "AlwaysTRUE" AND "IO_Valve_T04_Chili"."AV-04.03".FB_OPEN;
   "T-04_ChiliAwetan_3".IN_FBAV_Transfer := "AlwaysTRUE" AND (("T-04_ChiliAwetan_3".IN_Dose_Header_1 AND "IO_Valve_T04_Chili"."AV-04.12".FB_OPEN) OR ("T-04_ChiliAwetan_3".IN_Dose_Header_2 AND "IO_Valve_T04_Chili"."AV-04.11".FB_OPEN));
   "T-04_ChiliAwetan_3".IN_FBAV_CIP_Tank := "AlwaysTRUE" AND "IO_Valve_T02_Chili"."AV-02.20".FB_OPEN AND "IO_Valve_T04_Chili"."AV-04.02".FB_OPEN AND "IO_Valve_T04_Chili"."AV-04.04".FB_OPEN AND ("IO_Valve_T08_FreshChili"."AV-08.17".FB_OPEN OR "IO_Valve_T02_Chili"."AV-02.06".FB_OPEN);
   "T-04_ChiliAwetan_3".IN_FBAV_CIP_Line := "AlwaysTRUE" AND "IO_Valve_T02_Chili"."AV-02.20".FB_OPEN AND "IO_Valve_T04_Chili"."AV-04.01".FB_OPEN AND "IO_Valve_T04_Chili"."AV-04.05".FB_OPEN AND ("IO_Valve_T04_Chili"."AV-04.13".FB_OPEN OR "IO_Valve_T04_Chili"."AV-04.10".FB_OPEN);
   "T-04_ChiliAwetan_3".IN_FBP_Inload := "AlwaysTRUE" AND "IO Motor MCC Preparation_DB"."P-03.03".QRUN;
   IF "AlwaysTRUE" THEN
       "T-04_ChiliAwetan_3".IN_FBP_Inload_SP := "IO Motor MCC Preparation_DB"."P-03.03".QAct_Speed;
   END_IF;
   "T-04_ChiliAwetan_3".IN_FBP_Transfer := "AlwaysTRUE" AND "IO Motor MCC Preparation_DB"."P-04.01".QRUN;
   IF "AlwaysTRUE" THEN
       "T-04_ChiliAwetan_3".IN_FBP_Transfer_SP := "IO Motor MCC Preparation_DB"."P-04.01".QAct_Speed;
   END_IF;
   "T-04_ChiliAwetan_3".IN_FBP_CIP := "AlwaysTRUE" AND "IO Motor MCC Preparation_DB"."P-08.02".QRUN;
   IF "AlwaysTRUE" THEN
       "T-04_ChiliAwetan_3".IN_FBP_CIP_Sp := "IO Motor MCC Preparation_DB"."P-08.02".QAct_Speed;
   END_IF;
END_REGION

REGION Network 45: T-04.00 Comm to Blend
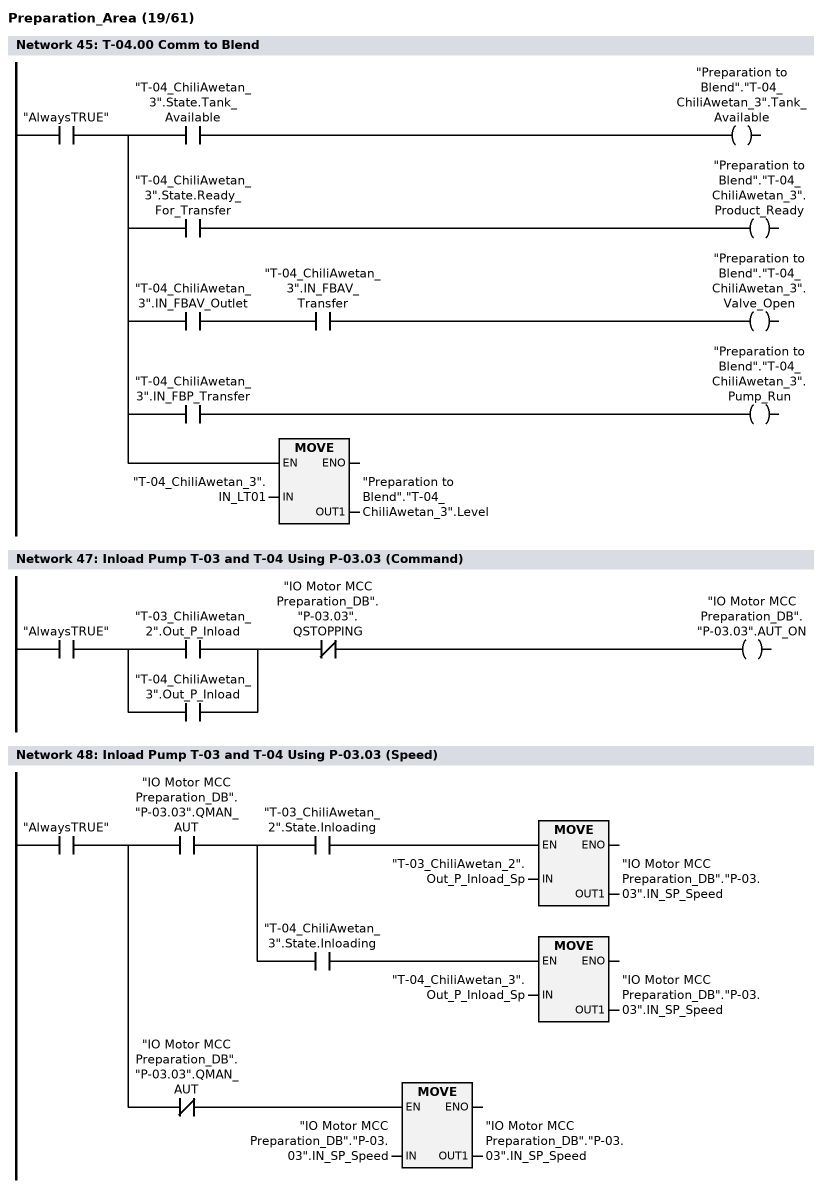
   RUNG wire#powerrail
      Contact( "AlwaysTRUE" )
      wire#w1
      Contact( "T-04_ChiliAwetan_3".State.Tank_Available )
      Coil( "Preparation to Blend"."T-04_ChiliAwetan_3".Tank_Available )
   END_RUNG
   RUNG wire#w1
      Contact( "T-04_ChiliAwetan_3".State.Ready_For_Transfer )
      Coil( "Preparation to Blend"."T-04_ChiliAwetan_3".Product_Ready )
   END_RUNG
   RUNG wire#w1
      Contact( "T-04_ChiliAwetan_3".IN_FBAV_Outlet )
      Contact( "T-04_ChiliAwetan_3".IN_FBAV_Transfer )
      Coil( "Preparation to Blend"."T-04_ChiliAwetan_3".Valve_Open )
   END_RUNG
   RUNG wire#w1
      Contact( "T-04_ChiliAwetan_3".IN_FBP_Transfer )
      Coil( "Preparation to Blend"."T-04_ChiliAwetan_3".Pump_Run )
   END_RUNG
   RUNG wire#w1
      Move(in := "T-04_ChiliAwetan_3".IN_LT01, out1 => "Preparation to Blend"."T-04_ChiliAwetan_3".Level)
   END_RUNG
   // the same network as SCL:
   "Preparation to Blend"."T-04_ChiliAwetan_3".Tank_Available := "AlwaysTRUE" AND "T-04_ChiliAwetan_3".State.Tank_Available;
   "Preparation to Blend"."T-04_ChiliAwetan_3".Product_Ready := "AlwaysTRUE" AND "T-04_ChiliAwetan_3".State.Ready_For_Transfer;
   "Preparation to Blend"."T-04_ChiliAwetan_3".Valve_Open := "AlwaysTRUE" AND "T-04_ChiliAwetan_3".IN_FBAV_Outlet AND "T-04_ChiliAwetan_3".IN_FBAV_Transfer;
   "Preparation to Blend"."T-04_ChiliAwetan_3".Pump_Run := "AlwaysTRUE" AND "T-04_ChiliAwetan_3".IN_FBP_Transfer;
   IF "AlwaysTRUE" THEN
       "Preparation to Blend"."T-04_ChiliAwetan_3".Level := "T-04_ChiliAwetan_3".IN_LT01;
   END_IF;
END_REGION

REGION Network 47: Inload Pump T-03 and T-04 Using P-03.03 (Command)
   RUNG wire#powerrail
      Contact( "AlwaysTRUE" )
      wire#w1
      Contact( "T-03_ChiliAwetan_2".Out_P_Inload )
      wire#w2
      I_Contact( "IO Motor MCC Preparation_DB"."P-03.03".QSTOPPING )
      Coil( "IO Motor MCC Preparation_DB"."P-03.03".AUT_ON )
   END_RUNG
   RUNG wire#w1
      Contact( "T-04_ChiliAwetan_3".Out_P_Inload )
   END_RUNG wire#w2
   // the same network as SCL:
   "IO Motor MCC Preparation_DB"."P-03.03".AUT_ON := "AlwaysTRUE" AND ("T-03_ChiliAwetan_2".Out_P_Inload OR "T-04_ChiliAwetan_3".Out_P_Inload) AND NOT "IO Motor MCC Preparation_DB"."P-03.03".QSTOPPING;
END_REGION

REGION Network 48: Inload Pump T-03 and T-04 Using P-03.03 (Speed)
   RUNG wire#powerrail
      Contact( "AlwaysTRUE" )
      wire#w1
      Contact( "IO Motor MCC Preparation_DB"."P-03.03".QMAN_AUT )
      wire#w2
      Contact( "T-03_ChiliAwetan_2".State.Inloading )
      Move(in := "T-03_ChiliAwetan_2".Out_P_Inload_Sp, out1 => "IO Motor MCC Preparation_DB"."P-03.03".IN_SP_Speed)
   END_RUNG
   RUNG wire#w2
      Contact( "T-04_ChiliAwetan_3".State.Inloading )
      Move(in := "T-04_ChiliAwetan_3".Out_P_Inload_Sp, out1 => "IO Motor MCC Preparation_DB"."P-03.03".IN_SP_Speed)
   END_RUNG
   RUNG wire#w1
      I_Contact( "IO Motor MCC Preparation_DB"."P-03.03".QMAN_AUT )
      Move(in := "IO Motor MCC Preparation_DB"."P-03.03".IN_SP_Speed, out1 => "IO Motor MCC Preparation_DB"."P-03.03".IN_SP_Speed)
   END_RUNG
   // the same network as SCL:
   #_w1 := "AlwaysTRUE" AND "IO Motor MCC Preparation_DB"."P-03.03".QMAN_AUT;
   IF #_w1 AND "T-03_ChiliAwetan_2".State.Inloading THEN
       "IO Motor MCC Preparation_DB"."P-03.03".IN_SP_Speed := "T-03_ChiliAwetan_2".Out_P_Inload_Sp;
   END_IF;
   IF #_w1 AND "T-04_ChiliAwetan_3".State.Inloading THEN
       "IO Motor MCC Preparation_DB"."P-03.03".IN_SP_Speed := "T-04_ChiliAwetan_3".Out_P_Inload_Sp;
   END_IF;
   IF "AlwaysTRUE" AND NOT "IO Motor MCC Preparation_DB"."P-03.03".QMAN_AUT THEN
       "IO Motor MCC Preparation_DB"."P-03.03".IN_SP_Speed := "IO Motor MCC Preparation_DB"."P-03.03".IN_SP_Speed;
   END_IF;
END_REGION

REGION Network 49: Comm T-03 and T-04 to Tipper 2
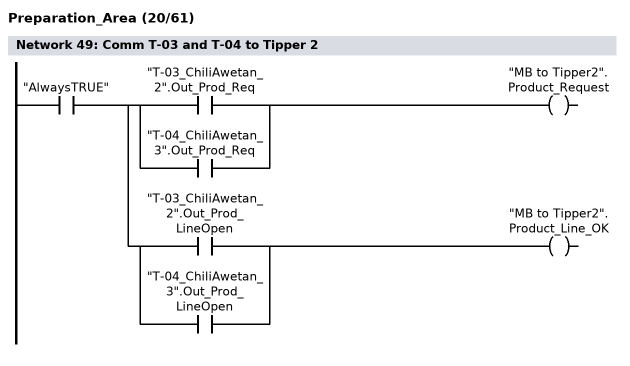
   RUNG wire#powerrail
      Contact( "AlwaysTRUE" )
      wire#w1
      Contact( "T-03_ChiliAwetan_2".Out_Prod_Req )
      wire#w2
      Coil( "MB to Tipper2".Product_Request )
   END_RUNG
   RUNG wire#w1
      Contact( "T-04_ChiliAwetan_3".Out_Prod_Req )
   END_RUNG wire#w2
   RUNG wire#w1
      Contact( "T-03_ChiliAwetan_2".Out_Prod_LineOpen )
      wire#w3
      Coil( "MB to Tipper2".Product_Line_OK )
   END_RUNG
   RUNG wire#w1
      Contact( "T-04_ChiliAwetan_3".Out_Prod_LineOpen )
   END_RUNG wire#w3
   // the same network as SCL:
   "MB to Tipper2".Product_Request := "AlwaysTRUE" AND ("T-03_ChiliAwetan_2".Out_Prod_Req OR "T-04_ChiliAwetan_3".Out_Prod_Req);
   "MB to Tipper2".Product_Line_OK := "AlwaysTRUE" AND ("T-03_ChiliAwetan_2".Out_Prod_LineOpen OR "T-04_ChiliAwetan_3".Out_Prod_LineOpen);
END_REGION

NETWORK
TITLE = T-05.00 DOSE ON OFF
      O     "Blend to Preparation"."T-20".Raw_Material.Tomato.DoseRun;
      O     "Blend to Preparation"."T-21".Raw_Material.Tomato.DoseRun;
      O     "Blend to Preparation"."T-30".Raw_Material.Tomato.DoseRun;
      O     "Blend to Preparation"."T-31".Raw_Material.Tomato.DoseRun;
      O     "Blend to Preparation"."T-40".Raw_Material.Tomato.DoseRun;
      O     "Blend to Preparation"."T-41".Raw_Material.Tomato.DoseRun;
      =     "T-05_Tomato".IN_Dose_Run;

NETWORK
TITLE = T-05.00 DOSE PAUSE
      O     "Blend to Preparation"."T-20".Raw_Material.Tomato.DoseHeld;
      O     "Blend to Preparation"."T-21".Raw_Material.Tomato.DoseHeld;
      O     "Blend to Preparation"."T-30".Raw_Material.Tomato.DoseHeld;
      O     "Blend to Preparation"."T-31".Raw_Material.Tomato.DoseHeld;
      O     "Blend to Preparation"."T-40".Raw_Material.Tomato.DoseHeld;
      O     "Blend to Preparation"."T-41".Raw_Material.Tomato.DoseHeld;
      =     "T-05_Tomato".IN_Dose_Held;

NETWORK
TITLE = T-05.00 DOSE VALVE CMD
      O(;
      A     "Blend to Preparation"."T-20".Raw_Material.Tomato.DoseRun;
      A     "Blend to Preparation"."T-20".Raw_Material.Tomato.ValveCMD;
      );
      O(;
      A     "Blend to Preparation"."T-21".Raw_Material.Tomato.DoseRun;
      A     "Blend to Preparation"."T-21".Raw_Material.Tomato.ValveCMD;
      );
      O(;
      A     "Blend to Preparation"."T-30".Raw_Material.Tomato.DoseRun;
      A     "Blend to Preparation"."T-30".Raw_Material.Tomato.ValveCMD;
      );
      O(;
      A     "Blend to Preparation"."T-31".Raw_Material.Tomato.DoseRun;
      A     "Blend to Preparation"."T-31".Raw_Material.Tomato.ValveCMD;
      );
      O(;
      A     "Blend to Preparation"."T-40".Raw_Material.Tomato.DoseRun;
      A     "Blend to Preparation"."T-40".Raw_Material.Tomato.ValveCMD;
      );
      O(;
      A     "Blend to Preparation"."T-41".Raw_Material.Tomato.DoseRun;
      A     "Blend to Preparation"."T-41".Raw_Material.Tomato.ValveCMD;
      );
      =     "T-05_Tomato".IN_Dose_Valve_Cmd;



NETWORK
TITLE = T-05.00 DOSE Pump CMD
      O(;
      A     "Blend to Preparation"."T-20".Raw_Material.Tomato.DoseRun;
      A     "Blend to Preparation"."T-20".Raw_Material.Tomato.PumpCMD;
      );
      O(;
      A     "Blend to Preparation"."T-21".Raw_Material.Tomato.DoseRun;
      A     "Blend to Preparation"."T-21".Raw_Material.Tomato.PumpCMD;
      );
      O(;
      A     "Blend to Preparation"."T-30".Raw_Material.Tomato.DoseRun;
      A     "Blend to Preparation"."T-30".Raw_Material.Tomato.PumpCMD;
      );
      O(;
      A     "Blend to Preparation"."T-31".Raw_Material.Tomato.DoseRun;
      A     "Blend to Preparation"."T-31".Raw_Material.Tomato.PumpCMD;
      );
      O(;
      A     "Blend to Preparation"."T-40".Raw_Material.Tomato.DoseRun;
      A     "Blend to Preparation"."T-40".Raw_Material.Tomato.PumpCMD;
      );
      O(;
      A     "Blend to Preparation"."T-41".Raw_Material.Tomato.DoseRun;
      A     "Blend to Preparation"."T-41".Raw_Material.Tomato.PumpCMD;
      );
      =     "T-05_Tomato".IN_Dose_Pump_Cmd;



NETWORK
TITLE = T-05.00 DOSE PUMP SPEED
// Checking
      O     "Blend to Preparation"."T-20".Raw_Material.Tomato.DoseRun;
      JC    SP_05_FROM_20;
      O     "Blend to Preparation"."T-21".Raw_Material.Tomato.DoseRun;
      JC    SP_05_FROM_21;
      O     "Blend to Preparation"."T-30".Raw_Material.Tomato.DoseRun;
      JC    SP_05_FROM_30;
      O     "Blend to Preparation"."T-31".Raw_Material.Tomato.DoseRun;
      JC    SP_05_FROM_31;
      O     "Blend to Preparation"."T-40".Raw_Material.Tomato.DoseRun;
      JC    SP_05_FROM_40;
      O     "Blend to Preparation"."T-41".Raw_Material.Tomato.DoseRun;
      JC    SP_05_FROM_41;
//Jump to end if Blend not Dosing
      JC    SP_05_SELF;
//Load Set Point
SP_05_FROM_20:L     "Blend to Preparation".Recipe."T-20".Tomato.SP_PumpSpeed;
      T     "T-05_Tomato".IN_Dose_Pump_Sp;
      JC    SP_05_SELF;
SP_05_FROM_21:L     "Blend to Preparation".Recipe."T-21".Tomato.SP_PumpSpeed;
      T     "T-05_Tomato".IN_Dose_Pump_Sp;
      JC    SP_05_SELF;
SP_05_FROM_30:L     "Blend to Preparation".Recipe."T-30".Tomato.SP_PumpSpeed;
      T     "T-05_Tomato".IN_Dose_Pump_Sp;
      JC    SP_05_SELF;
SP_05_FROM_31:L     "Blend to Preparation".Recipe."T-31".Tomato.SP_PumpSpeed;
      T     "T-05_Tomato".IN_Dose_Pump_Sp;
      JC    SP_05_SELF;
SP_05_FROM_40:L     "Blend to Preparation".Recipe."T-40".Tomato.SP_PumpSpeed;
      T     "T-05_Tomato".IN_Dose_Pump_Sp;
      JC    SP_05_SELF;
SP_05_FROM_41:L     "Blend to Preparation".Recipe."T-41".Tomato.SP_PumpSpeed;
      T     "T-05_Tomato".IN_Dose_Pump_Sp;
      JC    SP_05_SELF;
// END
SP_05_SELF:L     "T-05_Tomato".IN_Dose_Pump_Sp;
      T     "T-05_Tomato".IN_Dose_Pump_Sp;


NETWORK
TITLE = T-05.00 Header Req
// HEADER 1 Req
      O     "Blend to Preparation"."T-20".Raw_Material.Tomato.Header1_Req;
      O     "Blend to Preparation"."T-21".Raw_Material.Tomato.Header1_Req;
      O     "Blend to Preparation"."T-30".Raw_Material.Tomato.Header1_Req;
      O     "Blend to Preparation"."T-31".Raw_Material.Tomato.Header1_Req;
      O     "Blend to Preparation"."T-40".Raw_Material.Tomato.Header1_Req;
      O     "Blend to Preparation"."T-41".Raw_Material.Tomato.Header1_Req;
      =     "T-05_Tomato".IN_Dose_Header_1;

// HEADER 2 Req
      O     "Blend to Preparation"."T-20".Raw_Material.Tomato.Header2_Req;
      O     "Blend to Preparation"."T-21".Raw_Material.Tomato.Header2_Req;
      O     "Blend to Preparation"."T-30".Raw_Material.Tomato.Header2_Req;
      O     "Blend to Preparation"."T-31".Raw_Material.Tomato.Header2_Req;
      O     "Blend to Preparation"."T-40".Raw_Material.Tomato.Header2_Req;
      O     "Blend to Preparation"."T-41".Raw_Material.Tomato.Header2_Req;
      =     "T-05_Tomato".IN_Dose_Header_2;


REGION Network 57: T-05.00 LineTransferOK
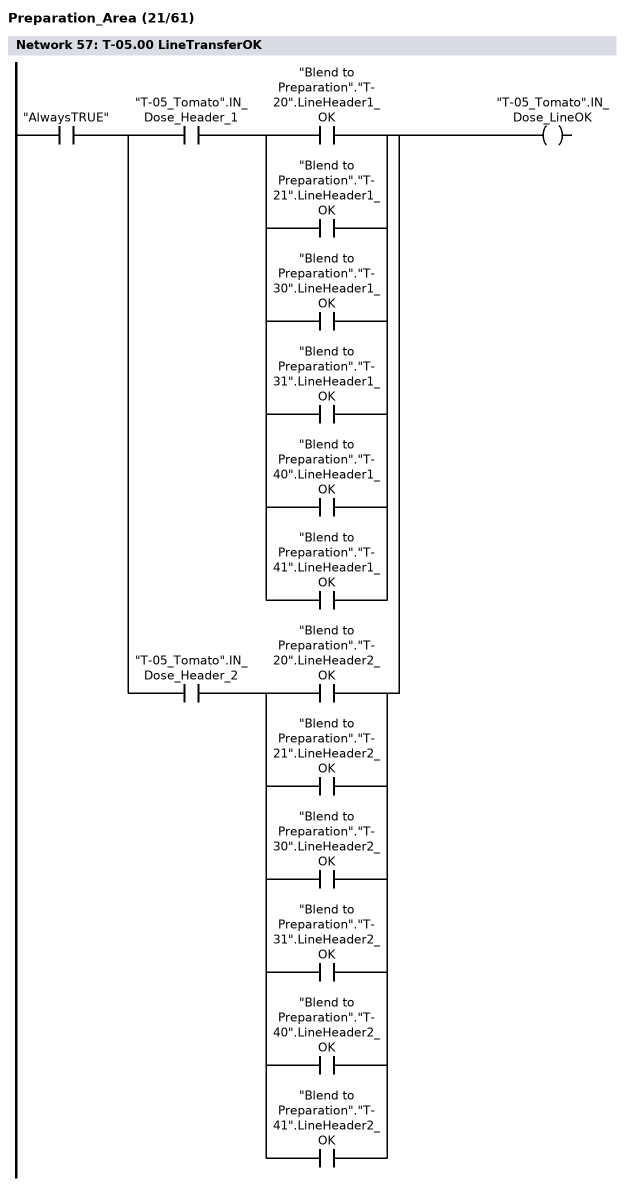
   RUNG wire#powerrail
      Contact( "AlwaysTRUE" )
      wire#w1
      Contact( "T-05_Tomato".IN_Dose_Header_1 )
      wire#w2
      Contact( "Blend to Preparation"."T-20".LineHeader1_OK )
      wire#w3
      Coil( "T-05_Tomato".IN_Dose_LineOK )
   END_RUNG
   RUNG wire#w2
      Contact( "Blend to Preparation"."T-21".LineHeader1_OK )
   END_RUNG wire#w3
   RUNG wire#w2
      Contact( "Blend to Preparation"."T-30".LineHeader1_OK )
   END_RUNG wire#w3
   RUNG wire#w2
      Contact( "Blend to Preparation"."T-31".LineHeader1_OK )
   END_RUNG wire#w3
   RUNG wire#w2
      Contact( "Blend to Preparation"."T-40".LineHeader1_OK )
   END_RUNG wire#w3
   RUNG wire#w2
      Contact( "Blend to Preparation"."T-41".LineHeader1_OK )
   END_RUNG wire#w3
   RUNG wire#w1
      Contact( "T-05_Tomato".IN_Dose_Header_2 )
      wire#w4
      Contact( "Blend to Preparation"."T-20".LineHeader2_OK )
   END_RUNG wire#w3
   RUNG wire#w4
      Contact( "Blend to Preparation"."T-21".LineHeader2_OK )
   END_RUNG wire#w3
   RUNG wire#w4
      Contact( "Blend to Preparation"."T-30".LineHeader2_OK )
   END_RUNG wire#w3
   RUNG wire#w4
      Contact( "Blend to Preparation"."T-31".LineHeader2_OK )
   END_RUNG wire#w3
   RUNG wire#w4
      Contact( "Blend to Preparation"."T-40".LineHeader2_OK )
   END_RUNG wire#w3
   RUNG wire#w4
      Contact( "Blend to Preparation"."T-41".LineHeader2_OK )
   END_RUNG wire#w3
   // the same network as SCL:
   "T-05_Tomato".IN_Dose_LineOK := "AlwaysTRUE" AND (("T-05_Tomato".IN_Dose_Header_1 AND ("Blend to Preparation"."T-20".LineHeader1_OK OR "Blend to Preparation"."T-21".LineHeader1_OK OR "Blend to Preparation"."T-30".LineHeader1_OK OR "Blend to Preparation"."T-31".LineHeader1_OK OR "Blend to Preparation"."T-40".LineHeader1_OK OR "Blend to Preparation"."T-41".LineHeader1_OK)) OR ("T-05_Tomato".IN_Dose_Header_2 AND ("Blend to Preparation"."T-20".LineHeader2_OK OR "Blend to Preparation"."T-21".LineHeader2_OK OR "Blend to Preparation"."T-30".LineHeader2_OK OR "Blend to Preparation"."T-31".LineHeader2_OK OR "Blend to Preparation"."T-40".LineHeader2_OK OR "Blend to Preparation"."T-41".LineHeader2_OK)));
END_REGION

REGION Network 58: T-05____Tomato
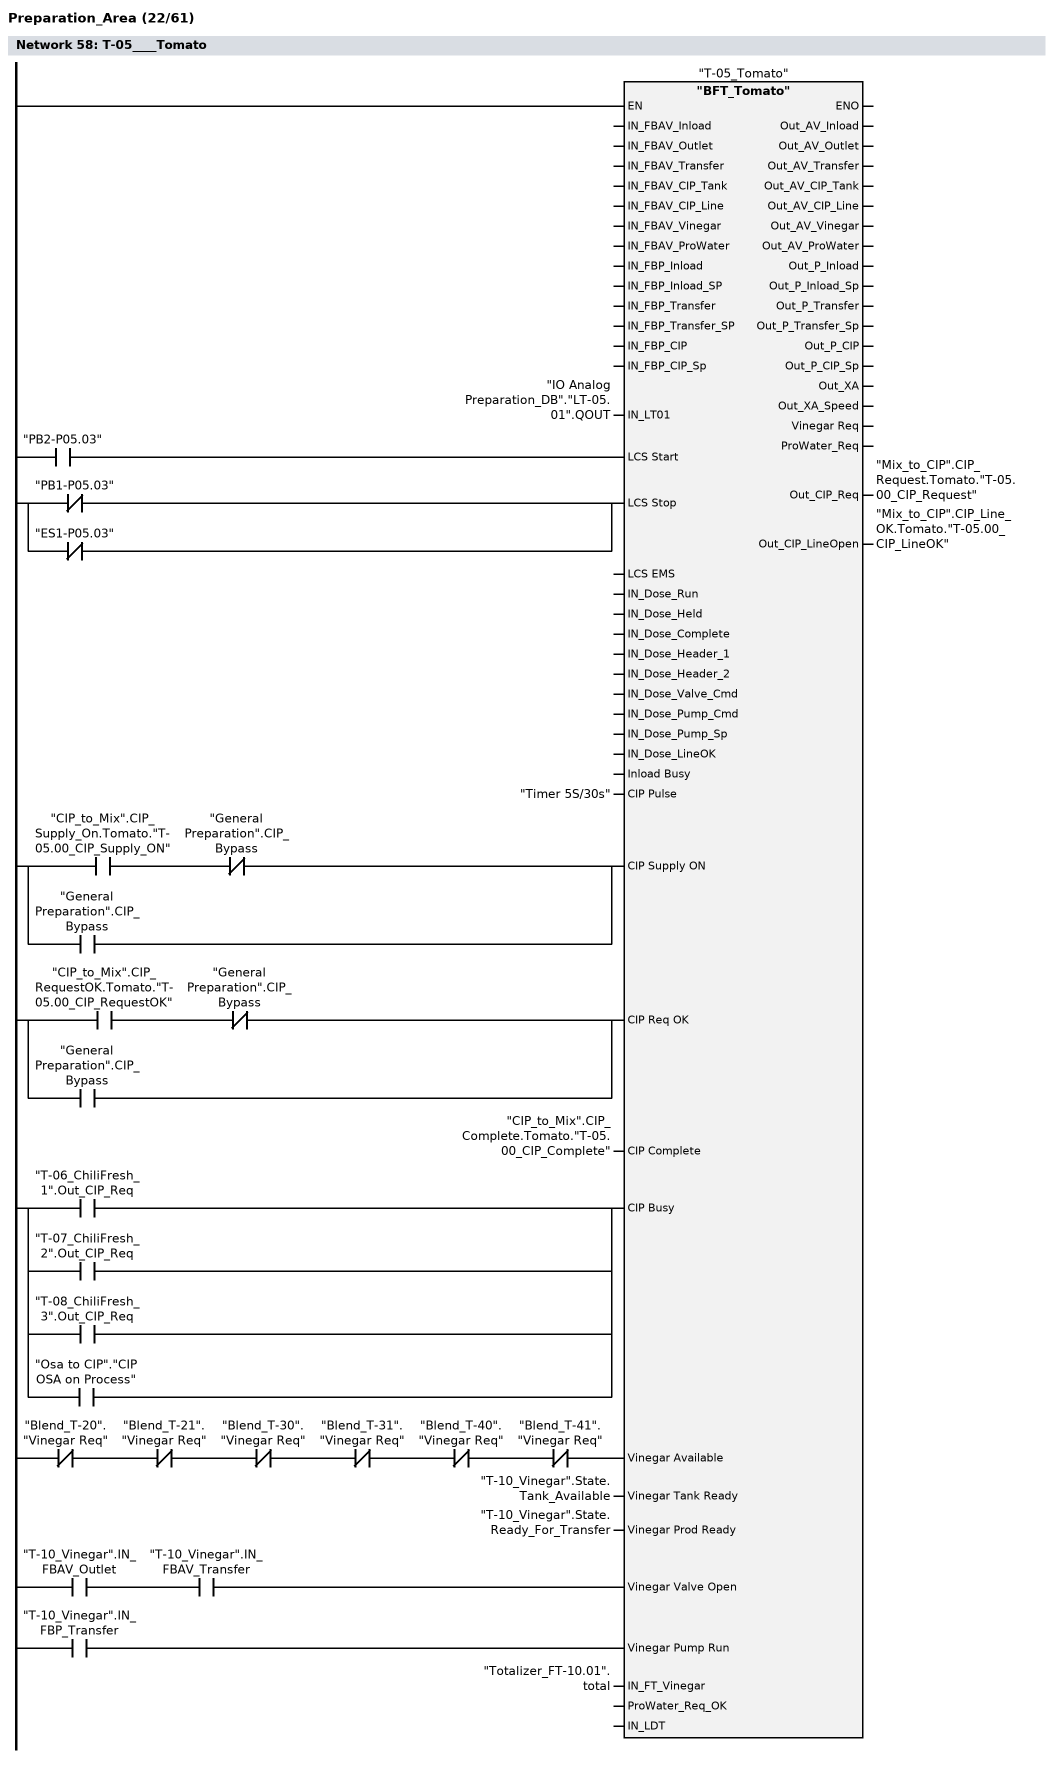
   RUNG wire#powerrail
      "T-05_Tomato"("LCS Start" := wire#w1, "LCS Stop" := wire#w2, "CIP Supply ON" := wire#w3, "CIP Req OK" := wire#w4, "CIP Busy" := wire#w5, "Vinegar Available" := wire#w6, "Vinegar Valve Open" := wire#w7, "Vinegar Pump Run" := wire#w8, IN_FBAV_Inload :=, IN_FBAV_Outlet :=, IN_FBAV_Transfer :=, IN_FBAV_CIP_Tank :=, IN_FBAV_CIP_Line :=, IN_FBAV_Vinegar :=, IN_FBAV_ProWater :=, IN_FBP_Inload :=, IN_FBP_Inload_SP :=, IN_FBP_Transfer :=, IN_FBP_Transfer_SP :=, IN_FBP_CIP :=, IN_FBP_CIP_Sp :=, IN_LT01 := "IO Analog Preparation_DB"."LT-05.01".QOUT, "LCS EMS" :=, IN_Dose_Run :=, IN_Dose_Held :=, IN_Dose_Complete :=, IN_Dose_Header_1 :=, IN_Dose_Header_2 :=, IN_Dose_Valve_Cmd :=, IN_Dose_Pump_Cmd :=, IN_Dose_Pump_Sp :=, IN_Dose_LineOK :=, "Inload Busy" :=, "CIP Pulse" := "Timer 5S/30s", "CIP Complete" := "CIP_to_Mix".CIP_Complete.Tomato."T-05.00_CIP_Complete", "Vinegar Tank Ready" := "T-10_Vinegar".State.Tank_Available, "Vinegar Prod Ready" := "T-10_Vinegar".State.Ready_For_Transfer, IN_FT_Vinegar := "Totalizer_FT-10.01".total, ProWater_Req_OK :=, IN_LDT :=, Out_AV_Inload =>, Out_AV_Outlet =>, Out_AV_Transfer =>, Out_AV_CIP_Tank =>, Out_AV_CIP_Line =>, Out_AV_Vinegar =>, Out_AV_ProWater =>, Out_P_Inload =>, Out_P_Inload_Sp =>, Out_P_Transfer =>, Out_P_Transfer_Sp =>, Out_P_CIP =>, Out_P_CIP_Sp =>, Out_XA =>, Out_XA_Speed =>, "Vinegar Req" =>, ProWater_Req =>, Out_CIP_Req => "Mix_to_CIP".CIP_Request.Tomato."T-05.00_CIP_Request", Out_CIP_LineOpen => "Mix_to_CIP".CIP_Line_OK.Tomato."T-05.00_CIP_LineOK")
   END_RUNG
   RUNG wire#powerrail
      Contact( "PB2-P05.03" )
   END_RUNG wire#w1
   RUNG wire#powerrail
      I_Contact( "PB1-P05.03" )
   END_RUNG wire#w2
   RUNG wire#powerrail
      I_Contact( "ES1-P05.03" )
   END_RUNG wire#w2
   RUNG wire#powerrail
      Contact( "CIP_to_Mix".CIP_Supply_On.Tomato."T-05.00_CIP_Supply_ON" )
      I_Contact( "General Preparation".CIP_Bypass )
   END_RUNG wire#w3
   RUNG wire#powerrail
      Contact( "General Preparation".CIP_Bypass )
   END_RUNG wire#w3
   RUNG wire#powerrail
      Contact( "CIP_to_Mix".CIP_RequestOK.Tomato."T-05.00_CIP_RequestOK" )
      I_Contact( "General Preparation".CIP_Bypass )
   END_RUNG wire#w4
   RUNG wire#powerrail
      Contact( "General Preparation".CIP_Bypass )
   END_RUNG wire#w4
   RUNG wire#powerrail
      Contact( "T-06_ChiliFresh_1".Out_CIP_Req )
   END_RUNG wire#w5
   RUNG wire#powerrail
      Contact( "T-07_ChiliFresh_2".Out_CIP_Req )
   END_RUNG wire#w5
   RUNG wire#powerrail
      Contact( "T-08_ChiliFresh_3".Out_CIP_Req )
   END_RUNG wire#w5
   RUNG wire#powerrail
      Contact( "Osa to CIP"."CIP OSA on Process" )
   END_RUNG wire#w5
   RUNG wire#powerrail
      I_Contact( "Blend_T-20"."Vinegar Req" )
      I_Contact( "Blend_T-21"."Vinegar Req" )
      I_Contact( "Blend_T-30"."Vinegar Req" )
      I_Contact( "Blend_T-31"."Vinegar Req" )
      I_Contact( "Blend_T-40"."Vinegar Req" )
      I_Contact( "Blend_T-41"."Vinegar Req" )
   END_RUNG wire#w6
   RUNG wire#powerrail
      Contact( "T-10_Vinegar".IN_FBAV_Outlet )
      Contact( "T-10_Vinegar".IN_FBAV_Transfer )
   END_RUNG wire#w7
   RUNG wire#powerrail
      Contact( "T-10_Vinegar".IN_FBP_Transfer )
   END_RUNG wire#w8
   // the same network as SCL:
   "T-05_Tomato"(IN_LT01 := "IO Analog Preparation_DB"."LT-05.01".QOUT,   // "BFT_Tomato"
                 "LCS Start" := "PB2-P05.03",
                 "LCS Stop" := NOT "PB1-P05.03" OR NOT "ES1-P05.03",
                 "CIP Pulse" := "Timer 5S/30s",
                 "CIP Supply ON" := ("CIP_to_Mix".CIP_Supply_On.Tomato."T-05.00_CIP_Supply_ON" AND NOT "General Preparation".CIP_Bypass) OR "General Preparation".CIP_Bypass,
                 "CIP Req OK" := ("CIP_to_Mix".CIP_RequestOK.Tomato."T-05.00_CIP_RequestOK" AND NOT "General Preparation".CIP_Bypass) OR "General Preparation".CIP_Bypass,
                 "CIP Complete" := "CIP_to_Mix".CIP_Complete.Tomato."T-05.00_CIP_Complete",
                 "CIP Busy" := "T-06_ChiliFresh_1".Out_CIP_Req OR "T-07_ChiliFresh_2".Out_CIP_Req OR "T-08_ChiliFresh_3".Out_CIP_Req OR "Osa to CIP"."CIP OSA on Process",
                 "Vinegar Available" := NOT "Blend_T-20"."Vinegar Req" AND NOT "Blend_T-21"."Vinegar Req" AND NOT "Blend_T-30"."Vinegar Req" AND NOT "Blend_T-31"."Vinegar Req" AND NOT "Blend_T-40"."Vinegar Req" AND NOT "Blend_T-41"."Vinegar Req",
                 "Vinegar Tank Ready" := "T-10_Vinegar".State.Tank_Available,
                 "Vinegar Prod Ready" := "T-10_Vinegar".State.Ready_For_Transfer,
                 "Vinegar Valve Open" := "T-10_Vinegar".IN_FBAV_Outlet AND "T-10_Vinegar".IN_FBAV_Transfer,
                 "Vinegar Pump Run" := "T-10_Vinegar".IN_FBP_Transfer,
                 IN_FT_Vinegar := "Totalizer_FT-10.01".total,
                 Out_CIP_Req => "Mix_to_CIP".CIP_Request.Tomato."T-05.00_CIP_Request",
                 Out_CIP_LineOpen => "Mix_to_CIP".CIP_Line_OK.Tomato."T-05.00_CIP_LineOK");
END_REGION

REGION Network 59: T-05.00 Valve Cmd
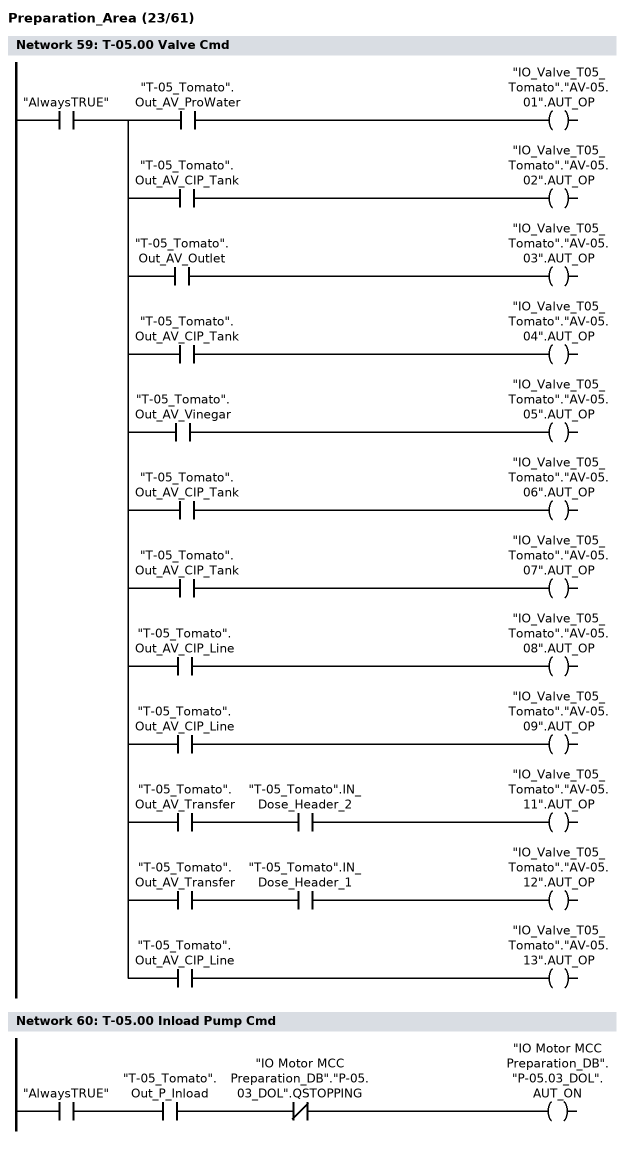
   RUNG wire#powerrail
      Contact( "AlwaysTRUE" )
      wire#w1
      Contact( "T-05_Tomato".Out_AV_ProWater )
      Coil( "IO_Valve_T05_Tomato"."AV-05.01".AUT_OP )
   END_RUNG
   RUNG wire#w1
      Contact( "T-05_Tomato".Out_AV_CIP_Tank )
      Coil( "IO_Valve_T05_Tomato"."AV-05.02".AUT_OP )
   END_RUNG
   RUNG wire#w1
      Contact( "T-05_Tomato".Out_AV_Outlet )
      Coil( "IO_Valve_T05_Tomato"."AV-05.03".AUT_OP )
   END_RUNG
   RUNG wire#w1
      Contact( "T-05_Tomato".Out_AV_CIP_Tank )
      Coil( "IO_Valve_T05_Tomato"."AV-05.04".AUT_OP )
   END_RUNG
   RUNG wire#w1
      Contact( "T-05_Tomato".Out_AV_Vinegar )
      Coil( "IO_Valve_T05_Tomato"."AV-05.05".AUT_OP )
   END_RUNG
   RUNG wire#w1
      Contact( "T-05_Tomato".Out_AV_CIP_Tank )
      Coil( "IO_Valve_T05_Tomato"."AV-05.06".AUT_OP )
   END_RUNG
   RUNG wire#w1
      Contact( "T-05_Tomato".Out_AV_CIP_Tank )
      Coil( "IO_Valve_T05_Tomato"."AV-05.07".AUT_OP )
   END_RUNG
   RUNG wire#w1
      Contact( "T-05_Tomato".Out_AV_CIP_Line )
      Coil( "IO_Valve_T05_Tomato"."AV-05.08".AUT_OP )
   END_RUNG
   RUNG wire#w1
      Contact( "T-05_Tomato".Out_AV_CIP_Line )
      Coil( "IO_Valve_T05_Tomato"."AV-05.09".AUT_OP )
   END_RUNG
   RUNG wire#w1
      Contact( "T-05_Tomato".Out_AV_Transfer )
      Contact( "T-05_Tomato".IN_Dose_Header_2 )
      Coil( "IO_Valve_T05_Tomato"."AV-05.11".AUT_OP )
   END_RUNG
   RUNG wire#w1
      Contact( "T-05_Tomato".Out_AV_Transfer )
      Contact( "T-05_Tomato".IN_Dose_Header_1 )
      Coil( "IO_Valve_T05_Tomato"."AV-05.12".AUT_OP )
   END_RUNG
   RUNG wire#w1
      Contact( "T-05_Tomato".Out_AV_CIP_Line )
      Coil( "IO_Valve_T05_Tomato"."AV-05.13".AUT_OP )
   END_RUNG
   // the same network as SCL:
   "IO_Valve_T05_Tomato"."AV-05.01".AUT_OP := "AlwaysTRUE" AND "T-05_Tomato".Out_AV_ProWater;
   "IO_Valve_T05_Tomato"."AV-05.02".AUT_OP := "AlwaysTRUE" AND "T-05_Tomato".Out_AV_CIP_Tank;
   "IO_Valve_T05_Tomato"."AV-05.03".AUT_OP := "AlwaysTRUE" AND "T-05_Tomato".Out_AV_Outlet;
   "IO_Valve_T05_Tomato"."AV-05.04".AUT_OP := "AlwaysTRUE" AND "T-05_Tomato".Out_AV_CIP_Tank;
   "IO_Valve_T05_Tomato"."AV-05.05".AUT_OP := "AlwaysTRUE" AND "T-05_Tomato".Out_AV_Vinegar;
   "IO_Valve_T05_Tomato"."AV-05.06".AUT_OP := "AlwaysTRUE" AND "T-05_Tomato".Out_AV_CIP_Tank;
   "IO_Valve_T05_Tomato"."AV-05.07".AUT_OP := "AlwaysTRUE" AND "T-05_Tomato".Out_AV_CIP_Tank;
   "IO_Valve_T05_Tomato"."AV-05.08".AUT_OP := "AlwaysTRUE" AND "T-05_Tomato".Out_AV_CIP_Line;
   "IO_Valve_T05_Tomato"."AV-05.09".AUT_OP := "AlwaysTRUE" AND "T-05_Tomato".Out_AV_CIP_Line;
   "IO_Valve_T05_Tomato"."AV-05.11".AUT_OP := "AlwaysTRUE" AND "T-05_Tomato".Out_AV_Transfer AND "T-05_Tomato".IN_Dose_Header_2;
   "IO_Valve_T05_Tomato"."AV-05.12".AUT_OP := "AlwaysTRUE" AND "T-05_Tomato".Out_AV_Transfer AND "T-05_Tomato".IN_Dose_Header_1;
   "IO_Valve_T05_Tomato"."AV-05.13".AUT_OP := "AlwaysTRUE" AND "T-05_Tomato".Out_AV_CIP_Line;
END_REGION

REGION Network 60: T-05.00 Inload Pump Cmd
   RUNG wire#powerrail
      Contact( "AlwaysTRUE" )
      Contact( "T-05_Tomato".Out_P_Inload )
      I_Contact( "IO Motor MCC Preparation_DB"."P-05.03_DOL".QSTOPPING )
      Coil( "IO Motor MCC Preparation_DB"."P-05.03_DOL".AUT_ON )
   END_RUNG
   // the same network as SCL:
   "IO Motor MCC Preparation_DB"."P-05.03_DOL".AUT_ON := "AlwaysTRUE" AND "T-05_Tomato".Out_P_Inload AND NOT "IO Motor MCC Preparation_DB"."P-05.03_DOL".QSTOPPING;
END_REGION

REGION Network 61: T-05.00 Transfer Pump Cmd and Speed
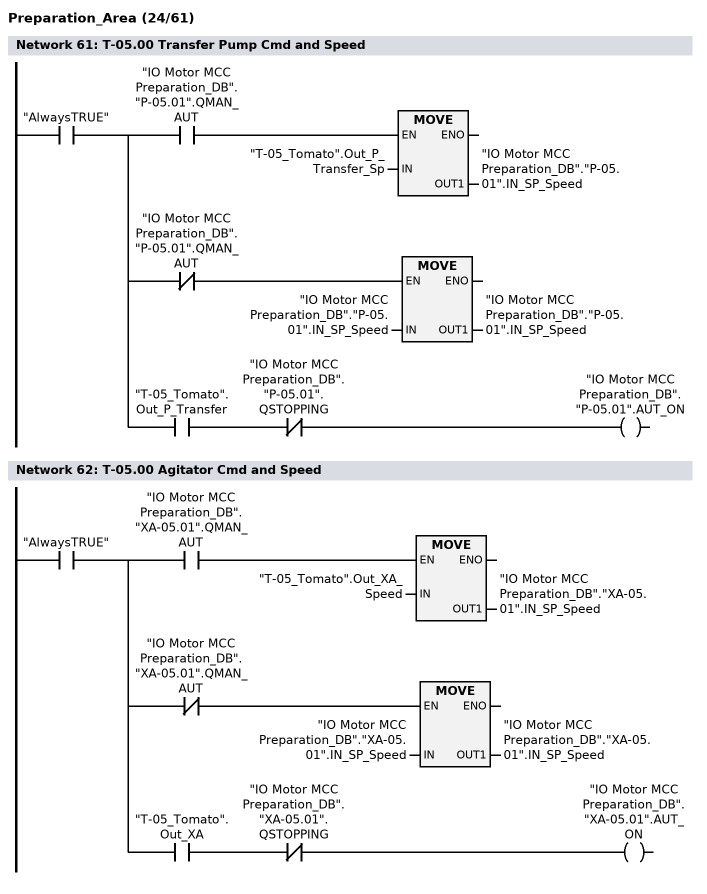
   RUNG wire#powerrail
      Contact( "AlwaysTRUE" )
      wire#w1
      Contact( "IO Motor MCC Preparation_DB"."P-05.01".QMAN_AUT )
      Move(in := "T-05_Tomato".Out_P_Transfer_Sp, out1 => "IO Motor MCC Preparation_DB"."P-05.01".IN_SP_Speed)
   END_RUNG
   RUNG wire#w1
      I_Contact( "IO Motor MCC Preparation_DB"."P-05.01".QMAN_AUT )
      Move(in := "IO Motor MCC Preparation_DB"."P-05.01".IN_SP_Speed, out1 => "IO Motor MCC Preparation_DB"."P-05.01".IN_SP_Speed)
   END_RUNG
   RUNG wire#w1
      Contact( "T-05_Tomato".Out_P_Transfer )
      I_Contact( "IO Motor MCC Preparation_DB"."P-05.01".QSTOPPING )
      Coil( "IO Motor MCC Preparation_DB"."P-05.01".AUT_ON )
   END_RUNG
   // the same network as SCL:
   IF "AlwaysTRUE" AND "IO Motor MCC Preparation_DB"."P-05.01".QMAN_AUT THEN
       "IO Motor MCC Preparation_DB"."P-05.01".IN_SP_Speed := "T-05_Tomato".Out_P_Transfer_Sp;
   END_IF;
   IF "AlwaysTRUE" AND NOT "IO Motor MCC Preparation_DB"."P-05.01".QMAN_AUT THEN
       "IO Motor MCC Preparation_DB"."P-05.01".IN_SP_Speed := "IO Motor MCC Preparation_DB"."P-05.01".IN_SP_Speed;
   END_IF;
   "IO Motor MCC Preparation_DB"."P-05.01".AUT_ON := "AlwaysTRUE" AND "T-05_Tomato".Out_P_Transfer AND NOT "IO Motor MCC Preparation_DB"."P-05.01".QSTOPPING;
END_REGION

REGION Network 62: T-05.00 Agitator Cmd and Speed
   RUNG wire#powerrail
      Contact( "AlwaysTRUE" )
      wire#w1
      Contact( "IO Motor MCC Preparation_DB"."XA-05.01".QMAN_AUT )
      Move(in := "T-05_Tomato".Out_XA_Speed, out1 => "IO Motor MCC Preparation_DB"."XA-05.01".IN_SP_Speed)
   END_RUNG
   RUNG wire#w1
      I_Contact( "IO Motor MCC Preparation_DB"."XA-05.01".QMAN_AUT )
      Move(in := "IO Motor MCC Preparation_DB"."XA-05.01".IN_SP_Speed, out1 => "IO Motor MCC Preparation_DB"."XA-05.01".IN_SP_Speed)
   END_RUNG
   RUNG wire#w1
      Contact( "T-05_Tomato".Out_XA )
      I_Contact( "IO Motor MCC Preparation_DB"."XA-05.01".QSTOPPING )
      Coil( "IO Motor MCC Preparation_DB"."XA-05.01".AUT_ON )
   END_RUNG
   // the same network as SCL:
   IF "AlwaysTRUE" AND "IO Motor MCC Preparation_DB"."XA-05.01".QMAN_AUT THEN
       "IO Motor MCC Preparation_DB"."XA-05.01".IN_SP_Speed := "T-05_Tomato".Out_XA_Speed;
   END_IF;
   IF "AlwaysTRUE" AND NOT "IO Motor MCC Preparation_DB"."XA-05.01".QMAN_AUT THEN
       "IO Motor MCC Preparation_DB"."XA-05.01".IN_SP_Speed := "IO Motor MCC Preparation_DB"."XA-05.01".IN_SP_Speed;
   END_IF;
   "IO Motor MCC Preparation_DB"."XA-05.01".AUT_ON := "AlwaysTRUE" AND "T-05_Tomato".Out_XA AND NOT "IO Motor MCC Preparation_DB"."XA-05.01".QSTOPPING;
END_REGION

REGION Network 63: T-05.00 Feedback Instrument
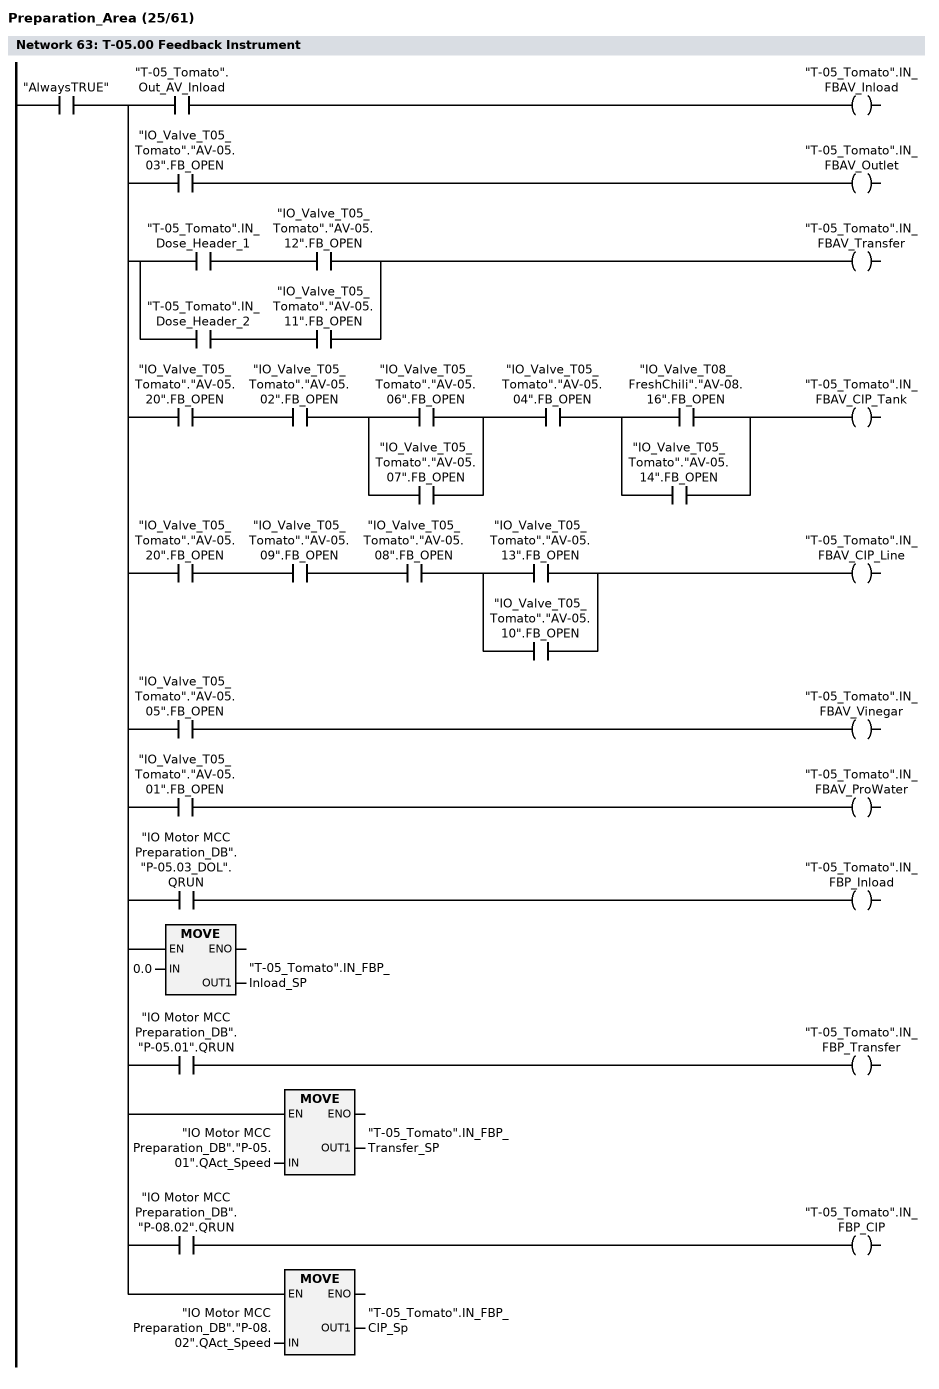
   RUNG wire#powerrail
      Contact( "AlwaysTRUE" )
      wire#w1
      Contact( "T-05_Tomato".Out_AV_Inload )
      Coil( "T-05_Tomato".IN_FBAV_Inload )
   END_RUNG
   RUNG wire#w1
      Contact( "IO_Valve_T05_Tomato"."AV-05.03".FB_OPEN )
      Coil( "T-05_Tomato".IN_FBAV_Outlet )
   END_RUNG
   RUNG wire#w1
      Contact( "T-05_Tomato".IN_Dose_Header_1 )
      Contact( "IO_Valve_T05_Tomato"."AV-05.12".FB_OPEN )
      wire#w2
      Coil( "T-05_Tomato".IN_FBAV_Transfer )
   END_RUNG
   RUNG wire#w1
      Contact( "T-05_Tomato".IN_Dose_Header_2 )
      Contact( "IO_Valve_T05_Tomato"."AV-05.11".FB_OPEN )
   END_RUNG wire#w2
   RUNG wire#w1
      Contact( "IO_Valve_T05_Tomato"."AV-05.20".FB_OPEN )
      Contact( "IO_Valve_T05_Tomato"."AV-05.02".FB_OPEN )
      wire#w3
      Contact( "IO_Valve_T05_Tomato"."AV-05.06".FB_OPEN )
      wire#w4
      Contact( "IO_Valve_T05_Tomato"."AV-05.04".FB_OPEN )
      wire#w5
      Contact( "IO_Valve_T08_FreshChili"."AV-08.16".FB_OPEN )
      wire#w6
      Coil( "T-05_Tomato".IN_FBAV_CIP_Tank )
   END_RUNG
   RUNG wire#w3
      Contact( "IO_Valve_T05_Tomato"."AV-05.07".FB_OPEN )
   END_RUNG wire#w4
   RUNG wire#w5
      Contact( "IO_Valve_T05_Tomato"."AV-05.14".FB_OPEN )
   END_RUNG wire#w6
   RUNG wire#w1
      Contact( "IO_Valve_T05_Tomato"."AV-05.20".FB_OPEN )
      Contact( "IO_Valve_T05_Tomato"."AV-05.09".FB_OPEN )
      Contact( "IO_Valve_T05_Tomato"."AV-05.08".FB_OPEN )
      wire#w7
      Contact( "IO_Valve_T05_Tomato"."AV-05.13".FB_OPEN )
      wire#w8
      Coil( "T-05_Tomato".IN_FBAV_CIP_Line )
   END_RUNG
   RUNG wire#w7
      Contact( "IO_Valve_T05_Tomato"."AV-05.10".FB_OPEN )
   END_RUNG wire#w8
   RUNG wire#w1
      Contact( "IO_Valve_T05_Tomato"."AV-05.05".FB_OPEN )
      Coil( "T-05_Tomato".IN_FBAV_Vinegar )
   END_RUNG
   RUNG wire#w1
      Contact( "IO_Valve_T05_Tomato"."AV-05.01".FB_OPEN )
      Coil( "T-05_Tomato".IN_FBAV_ProWater )
   END_RUNG
   RUNG wire#w1
      Contact( "IO Motor MCC Preparation_DB"."P-05.03_DOL".QRUN )
      Coil( "T-05_Tomato".IN_FBP_Inload )
   END_RUNG
   RUNG wire#w1
      Move(in := 0.0, out1 => "T-05_Tomato".IN_FBP_Inload_SP)
   END_RUNG
   RUNG wire#w1
      Contact( "IO Motor MCC Preparation_DB"."P-05.01".QRUN )
      Coil( "T-05_Tomato".IN_FBP_Transfer )
   END_RUNG
   RUNG wire#w1
      Move(in := "IO Motor MCC Preparation_DB"."P-05.01".QAct_Speed, out1 => "T-05_Tomato".IN_FBP_Transfer_SP)
   END_RUNG
   RUNG wire#w1
      Contact( "IO Motor MCC Preparation_DB"."P-08.02".QRUN )
      Coil( "T-05_Tomato".IN_FBP_CIP )
   END_RUNG
   RUNG wire#w1
      Move(in := "IO Motor MCC Preparation_DB"."P-08.02".QAct_Speed, out1 => "T-05_Tomato".IN_FBP_CIP_Sp)
   END_RUNG
   // the same network as SCL:
   "T-05_Tomato".IN_FBAV_Inload := "AlwaysTRUE" AND "T-05_Tomato".Out_AV_Inload;
   "T-05_Tomato".IN_FBAV_Outlet := "AlwaysTRUE" AND "IO_Valve_T05_Tomato"."AV-05.03".FB_OPEN;
   "T-05_Tomato".IN_FBAV_Transfer := "AlwaysTRUE" AND (("T-05_Tomato".IN_Dose_Header_1 AND "IO_Valve_T05_Tomato"."AV-05.12".FB_OPEN) OR ("T-05_Tomato".IN_Dose_Header_2 AND "IO_Valve_T05_Tomato"."AV-05.11".FB_OPEN));
   "T-05_Tomato".IN_FBAV_CIP_Tank := "AlwaysTRUE" AND "IO_Valve_T05_Tomato"."AV-05.20".FB_OPEN AND "IO_Valve_T05_Tomato"."AV-05.02".FB_OPEN AND ("IO_Valve_T05_Tomato"."AV-05.06".FB_OPEN OR "IO_Valve_T05_Tomato"."AV-05.07".FB_OPEN) AND "IO_Valve_T05_Tomato"."AV-05.04".FB_OPEN AND ("IO_Valve_T08_FreshChili"."AV-08.16".FB_OPEN OR "IO_Valve_T05_Tomato"."AV-05.14".FB_OPEN);
   "T-05_Tomato".IN_FBAV_CIP_Line := "AlwaysTRUE" AND "IO_Valve_T05_Tomato"."AV-05.20".FB_OPEN AND "IO_Valve_T05_Tomato"."AV-05.09".FB_OPEN AND "IO_Valve_T05_Tomato"."AV-05.08".FB_OPEN AND ("IO_Valve_T05_Tomato"."AV-05.13".FB_OPEN OR "IO_Valve_T05_Tomato"."AV-05.10".FB_OPEN);
   "T-05_Tomato".IN_FBAV_Vinegar := "AlwaysTRUE" AND "IO_Valve_T05_Tomato"."AV-05.05".FB_OPEN;
   "T-05_Tomato".IN_FBAV_ProWater := "AlwaysTRUE" AND "IO_Valve_T05_Tomato"."AV-05.01".FB_OPEN;
   "T-05_Tomato".IN_FBP_Inload := "AlwaysTRUE" AND "IO Motor MCC Preparation_DB"."P-05.03_DOL".QRUN;
   IF "AlwaysTRUE" THEN "T-05_Tomato".IN_FBP_Inload_SP := 0.0; END_IF;
   "T-05_Tomato".IN_FBP_Transfer := "AlwaysTRUE" AND "IO Motor MCC Preparation_DB"."P-05.01".QRUN;
   IF "AlwaysTRUE" THEN
       "T-05_Tomato".IN_FBP_Transfer_SP := "IO Motor MCC Preparation_DB"."P-05.01".QAct_Speed;
   END_IF;
   "T-05_Tomato".IN_FBP_CIP := "AlwaysTRUE" AND "IO Motor MCC Preparation_DB"."P-08.02".QRUN;
   IF "AlwaysTRUE" THEN
       "T-05_Tomato".IN_FBP_CIP_Sp := "IO Motor MCC Preparation_DB"."P-08.02".QAct_Speed;
   END_IF;
END_REGION

REGION Network 64: T-05.00 Comm to Blend
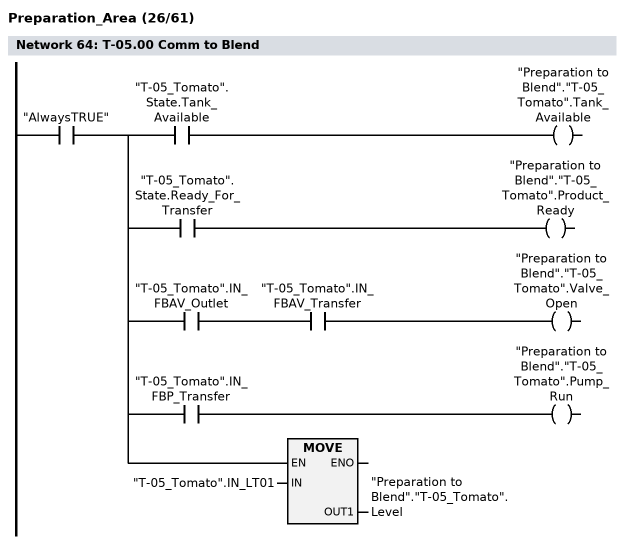
   RUNG wire#powerrail
      Contact( "AlwaysTRUE" )
      wire#w1
      Contact( "T-05_Tomato".State.Tank_Available )
      Coil( "Preparation to Blend"."T-05_Tomato".Tank_Available )
   END_RUNG
   RUNG wire#w1
      Contact( "T-05_Tomato".State.Ready_For_Transfer )
      Coil( "Preparation to Blend"."T-05_Tomato".Product_Ready )
   END_RUNG
   RUNG wire#w1
      Contact( "T-05_Tomato".IN_FBAV_Outlet )
      Contact( "T-05_Tomato".IN_FBAV_Transfer )
      Coil( "Preparation to Blend"."T-05_Tomato".Valve_Open )
   END_RUNG
   RUNG wire#w1
      Contact( "T-05_Tomato".IN_FBP_Transfer )
      Coil( "Preparation to Blend"."T-05_Tomato".Pump_Run )
   END_RUNG
   RUNG wire#w1
      Move(in := "T-05_Tomato".IN_LT01, out1 => "Preparation to Blend"."T-05_Tomato".Level)
   END_RUNG
   // the same network as SCL:
   "Preparation to Blend"."T-05_Tomato".Tank_Available := "AlwaysTRUE" AND "T-05_Tomato".State.Tank_Available;
   "Preparation to Blend"."T-05_Tomato".Product_Ready := "AlwaysTRUE" AND "T-05_Tomato".State.Ready_For_Transfer;
   "Preparation to Blend"."T-05_Tomato".Valve_Open := "AlwaysTRUE" AND "T-05_Tomato".IN_FBAV_Outlet AND "T-05_Tomato".IN_FBAV_Transfer;
   "Preparation to Blend"."T-05_Tomato".Pump_Run := "AlwaysTRUE" AND "T-05_Tomato".IN_FBP_Transfer;
   IF "AlwaysTRUE" THEN "Preparation to Blend"."T-05_Tomato".Level := "T-05_Tomato".IN_LT01; END_IF;
END_REGION

NETWORK
TITLE = T-06.00 DOSE ON OFF
      O     "Blend to Preparation"."T-20".Raw_Material.ChiliFresh_1.DoseRun;
      O     "Blend to Preparation"."T-21".Raw_Material.ChiliFresh_1.DoseRun;
      O     "Blend to Preparation"."T-30".Raw_Material.ChiliFresh_1.DoseRun;
      O     "Blend to Preparation"."T-31".Raw_Material.ChiliFresh_1.DoseRun;
      O     "Blend to Preparation"."T-40".Raw_Material.ChiliFresh_1.DoseRun;
      O     "Blend to Preparation"."T-41".Raw_Material.ChiliFresh_1.DoseRun;
      =     "T-06_ChiliFresh_1".IN_Dose_Run;

NETWORK
TITLE = T-06.00 DOSE PAUSE
      O     "Blend to Preparation"."T-20".Raw_Material.ChiliFresh_1.DoseHeld;
      O     "Blend to Preparation"."T-21".Raw_Material.ChiliFresh_1.DoseHeld;
      O     "Blend to Preparation"."T-30".Raw_Material.ChiliFresh_1.DoseHeld;
      O     "Blend to Preparation"."T-31".Raw_Material.ChiliFresh_1.DoseHeld;
      O     "Blend to Preparation"."T-40".Raw_Material.ChiliFresh_1.DoseHeld;
      O     "Blend to Preparation"."T-41".Raw_Material.ChiliFresh_1.DoseHeld;
      =     "T-06_ChiliFresh_1".IN_Dose_Held;

NETWORK
TITLE = T-06.00 DOSE VALVE CMD
      O(;
      A     "Blend to Preparation"."T-20".Raw_Material.ChiliFresh_1.DoseRun;
      A     "Blend to Preparation"."T-20".Raw_Material.ChiliFresh_1.ValveCMD;
      );
      O(;
      A     "Blend to Preparation"."T-21".Raw_Material.ChiliFresh_1.DoseRun;
      A     "Blend to Preparation"."T-21".Raw_Material.ChiliFresh_1.ValveCMD;
      );
      O(;
      A     "Blend to Preparation"."T-30".Raw_Material.ChiliFresh_1.DoseRun;
      A     "Blend to Preparation"."T-30".Raw_Material.ChiliFresh_1.ValveCMD;
      );
      O(;
      A     "Blend to Preparation"."T-31".Raw_Material.ChiliFresh_1.DoseRun;
      A     "Blend to Preparation"."T-31".Raw_Material.ChiliFresh_1.ValveCMD;
      );
      O(;
      A     "Blend to Preparation"."T-40".Raw_Material.ChiliFresh_1.DoseRun;
      A     "Blend to Preparation"."T-40".Raw_Material.ChiliFresh_1.ValveCMD;
      );
      O(;
      A     "Blend to Preparation"."T-41".Raw_Material.ChiliFresh_1.DoseRun;
      A     "Blend to Preparation"."T-41".Raw_Material.ChiliFresh_1.ValveCMD;
      );
      =     "T-06_ChiliFresh_1".IN_Dose_Valve_Cmd;



NETWORK
TITLE = T-06.00 DOSE Pump CMD
      O(;
      A     "Blend to Preparation"."T-20".Raw_Material.ChiliFresh_1.DoseRun;
      A     "Blend to Preparation"."T-20".Raw_Material.ChiliFresh_1.PumpCMD;
      );
      O(;
      A     "Blend to Preparation"."T-21".Raw_Material.ChiliFresh_1.DoseRun;
      A     "Blend to Preparation"."T-21".Raw_Material.ChiliFresh_1.PumpCMD;
      );
      O(;
      A     "Blend to Preparation"."T-30".Raw_Material.ChiliFresh_1.DoseRun;
      A     "Blend to Preparation"."T-30".Raw_Material.ChiliFresh_1.PumpCMD;
      );
      O(;
      A     "Blend to Preparation"."T-31".Raw_Material.ChiliFresh_1.DoseRun;
      A     "Blend to Preparation"."T-31".Raw_Material.ChiliFresh_1.PumpCMD;
      );
      O(;
      A     "Blend to Preparation"."T-40".Raw_Material.ChiliFresh_1.DoseRun;
      A     "Blend to Preparation"."T-40".Raw_Material.ChiliFresh_1.PumpCMD;
      );
      O(;
      A     "Blend to Preparation"."T-41".Raw_Material.ChiliFresh_1.DoseRun;
      A     "Blend to Preparation"."T-41".Raw_Material.ChiliFresh_1.PumpCMD;
      );
      =     "T-06_ChiliFresh_1".IN_Dose_Pump_Cmd;



NETWORK
TITLE = T-06.00 DOSE PUMP SPEED
// Checking
      O     "Blend to Preparation"."T-20".Raw_Material.ChiliFresh_1.DoseRun;
      JC    SP_06_FROM_20;
      O     "Blend to Preparation"."T-21".Raw_Material.ChiliFresh_1.DoseRun;
      JC    SP_06_FROM_21;
      O     "Blend to Preparation"."T-30".Raw_Material.ChiliFresh_1.DoseRun;
      JC    SP_06_FROM_30;
      O     "Blend to Preparation"."T-31".Raw_Material.ChiliFresh_1.DoseRun;
      JC    SP_06_FROM_31;
      O     "Blend to Preparation"."T-40".Raw_Material.ChiliFresh_1.DoseRun;
      JC    SP_06_FROM_40;
      O     "Blend to Preparation"."T-41".Raw_Material.ChiliFresh_1.DoseRun;
      JC    SP_06_FROM_41;
//Jump to end if Blend not Dosing
      JC    SP_06_SELF;
//Load Set Point
SP_06_FROM_20:L     "Blend to Preparation".Recipe."T-20".ChiliFresh_1.SP_PumpSpeed;
      T     "T-06_ChiliFresh_1".IN_Dose_Pump_Sp;
      JC    SP_06_SELF;
SP_06_FROM_21:L     "Blend to Preparation".Recipe."T-21".ChiliFresh_1.SP_PumpSpeed;
      T     "T-06_ChiliFresh_1".IN_Dose_Pump_Sp;
      JC    SP_06_SELF;
SP_06_FROM_30:L     "Blend to Preparation".Recipe."T-30".ChiliFresh_1.SP_PumpSpeed;
      T     "T-06_ChiliFresh_1".IN_Dose_Pump_Sp;
      JC    SP_06_SELF;
SP_06_FROM_31:L     "Blend to Preparation".Recipe."T-31".ChiliFresh_1.SP_PumpSpeed;
      T     "T-06_ChiliFresh_1".IN_Dose_Pump_Sp;
      JC    SP_06_SELF;
SP_06_FROM_40:L     "Blend to Preparation".Recipe."T-40".ChiliFresh_1.SP_PumpSpeed;
      T     "T-06_ChiliFresh_1".IN_Dose_Pump_Sp;
      JC    SP_06_SELF;
SP_06_FROM_41:L     "Blend to Preparation".Recipe."T-41".ChiliFresh_1.SP_PumpSpeed;
      T     "T-06_ChiliFresh_1".IN_Dose_Pump_Sp;
      JC    SP_06_SELF;
// END
SP_06_SELF:L     "T-06_ChiliFresh_1".IN_Dose_Pump_Sp;
      T     "T-06_ChiliFresh_1".IN_Dose_Pump_Sp;


NETWORK
TITLE = T-06.00 Header Req
// HEADER 1 Req
      O     "Blend to Preparation"."T-20".Raw_Material.ChiliFresh_1.Header1_Req;
      O     "Blend to Preparation"."T-21".Raw_Material.ChiliFresh_1.Header1_Req;
      O     "Blend to Preparation"."T-30".Raw_Material.ChiliFresh_1.Header1_Req;
      O     "Blend to Preparation"."T-31".Raw_Material.ChiliFresh_1.Header1_Req;
      O     "Blend to Preparation"."T-40".Raw_Material.ChiliFresh_1.Header1_Req;
      O     "Blend to Preparation"."T-41".Raw_Material.ChiliFresh_1.Header1_Req;
      =     "T-06_ChiliFresh_1".IN_Dose_Header_1;

// HEADER 2 Req
      O     "Blend to Preparation"."T-20".Raw_Material.ChiliFresh_1.Header2_Req;
      O     "Blend to Preparation"."T-21".Raw_Material.ChiliFresh_1.Header2_Req;
      O     "Blend to Preparation"."T-30".Raw_Material.ChiliFresh_1.Header2_Req;
      O     "Blend to Preparation"."T-31".Raw_Material.ChiliFresh_1.Header2_Req;
      O     "Blend to Preparation"."T-40".Raw_Material.ChiliFresh_1.Header2_Req;
      O     "Blend to Preparation"."T-41".Raw_Material.ChiliFresh_1.Header2_Req;
      =     "T-06_ChiliFresh_1".IN_Dose_Header_2;


REGION Network 73: T-06.00 LineTransferOK
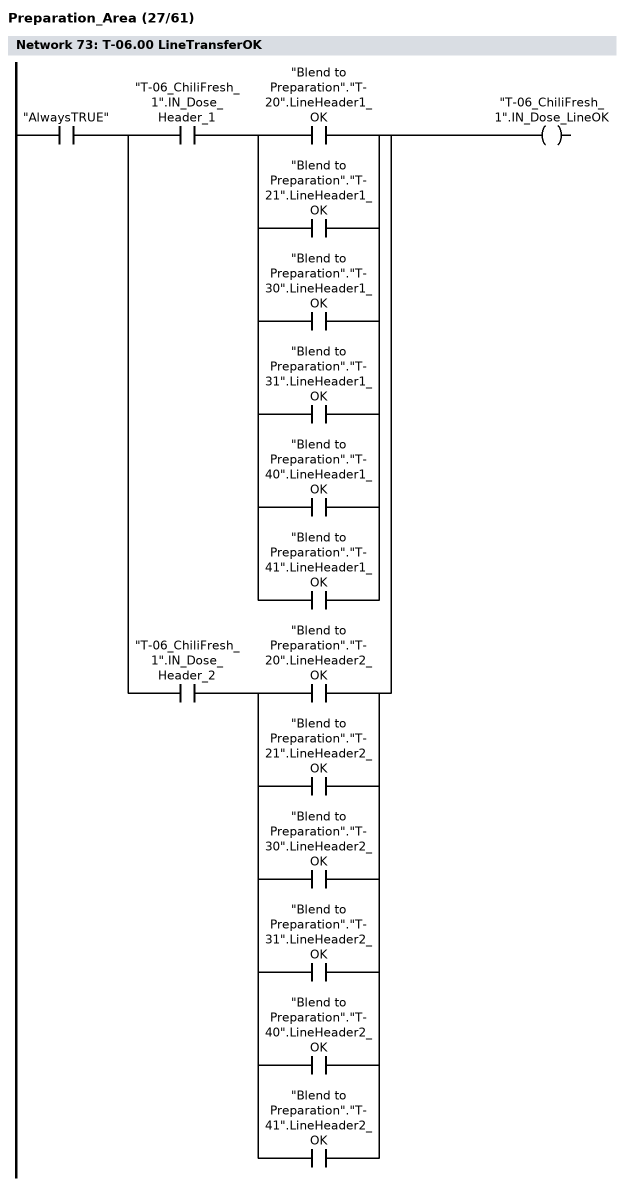
   RUNG wire#powerrail
      Contact( "AlwaysTRUE" )
      wire#w1
      Contact( "T-06_ChiliFresh_1".IN_Dose_Header_1 )
      wire#w2
      Contact( "Blend to Preparation"."T-20".LineHeader1_OK )
      wire#w3
      Coil( "T-06_ChiliFresh_1".IN_Dose_LineOK )
   END_RUNG
   RUNG wire#w2
      Contact( "Blend to Preparation"."T-21".LineHeader1_OK )
   END_RUNG wire#w3
   RUNG wire#w2
      Contact( "Blend to Preparation"."T-30".LineHeader1_OK )
   END_RUNG wire#w3
   RUNG wire#w2
      Contact( "Blend to Preparation"."T-31".LineHeader1_OK )
   END_RUNG wire#w3
   RUNG wire#w2
      Contact( "Blend to Preparation"."T-40".LineHeader1_OK )
   END_RUNG wire#w3
   RUNG wire#w2
      Contact( "Blend to Preparation"."T-41".LineHeader1_OK )
   END_RUNG wire#w3
   RUNG wire#w1
      Contact( "T-06_ChiliFresh_1".IN_Dose_Header_2 )
      wire#w4
      Contact( "Blend to Preparation"."T-20".LineHeader2_OK )
   END_RUNG wire#w3
   RUNG wire#w4
      Contact( "Blend to Preparation"."T-21".LineHeader2_OK )
   END_RUNG wire#w3
   RUNG wire#w4
      Contact( "Blend to Preparation"."T-30".LineHeader2_OK )
   END_RUNG wire#w3
   RUNG wire#w4
      Contact( "Blend to Preparation"."T-31".LineHeader2_OK )
   END_RUNG wire#w3
   RUNG wire#w4
      Contact( "Blend to Preparation"."T-40".LineHeader2_OK )
   END_RUNG wire#w3
   RUNG wire#w4
      Contact( "Blend to Preparation"."T-41".LineHeader2_OK )
   END_RUNG wire#w3
   // the same network as SCL:
   "T-06_ChiliFresh_1".IN_Dose_LineOK := "AlwaysTRUE" AND (("T-06_ChiliFresh_1".IN_Dose_Header_1 AND ("Blend to Preparation"."T-20".LineHeader1_OK OR "Blend to Preparation"."T-21".LineHeader1_OK OR "Blend to Preparation"."T-30".LineHeader1_OK OR "Blend to Preparation"."T-31".LineHeader1_OK OR "Blend to Preparation"."T-40".LineHeader1_OK OR "Blend to Preparation"."T-41".LineHeader1_OK)) OR ("T-06_ChiliFresh_1".IN_Dose_Header_2 AND ("Blend to Preparation"."T-20".LineHeader2_OK OR "Blend to Preparation"."T-21".LineHeader2_OK OR "Blend to Preparation"."T-30".LineHeader2_OK OR "Blend to Preparation"."T-31".LineHeader2_OK OR "Blend to Preparation"."T-40".LineHeader2_OK OR "Blend to Preparation"."T-41".LineHeader2_OK)));
END_REGION

REGION Network 74: T-06____Chili Fresh 1
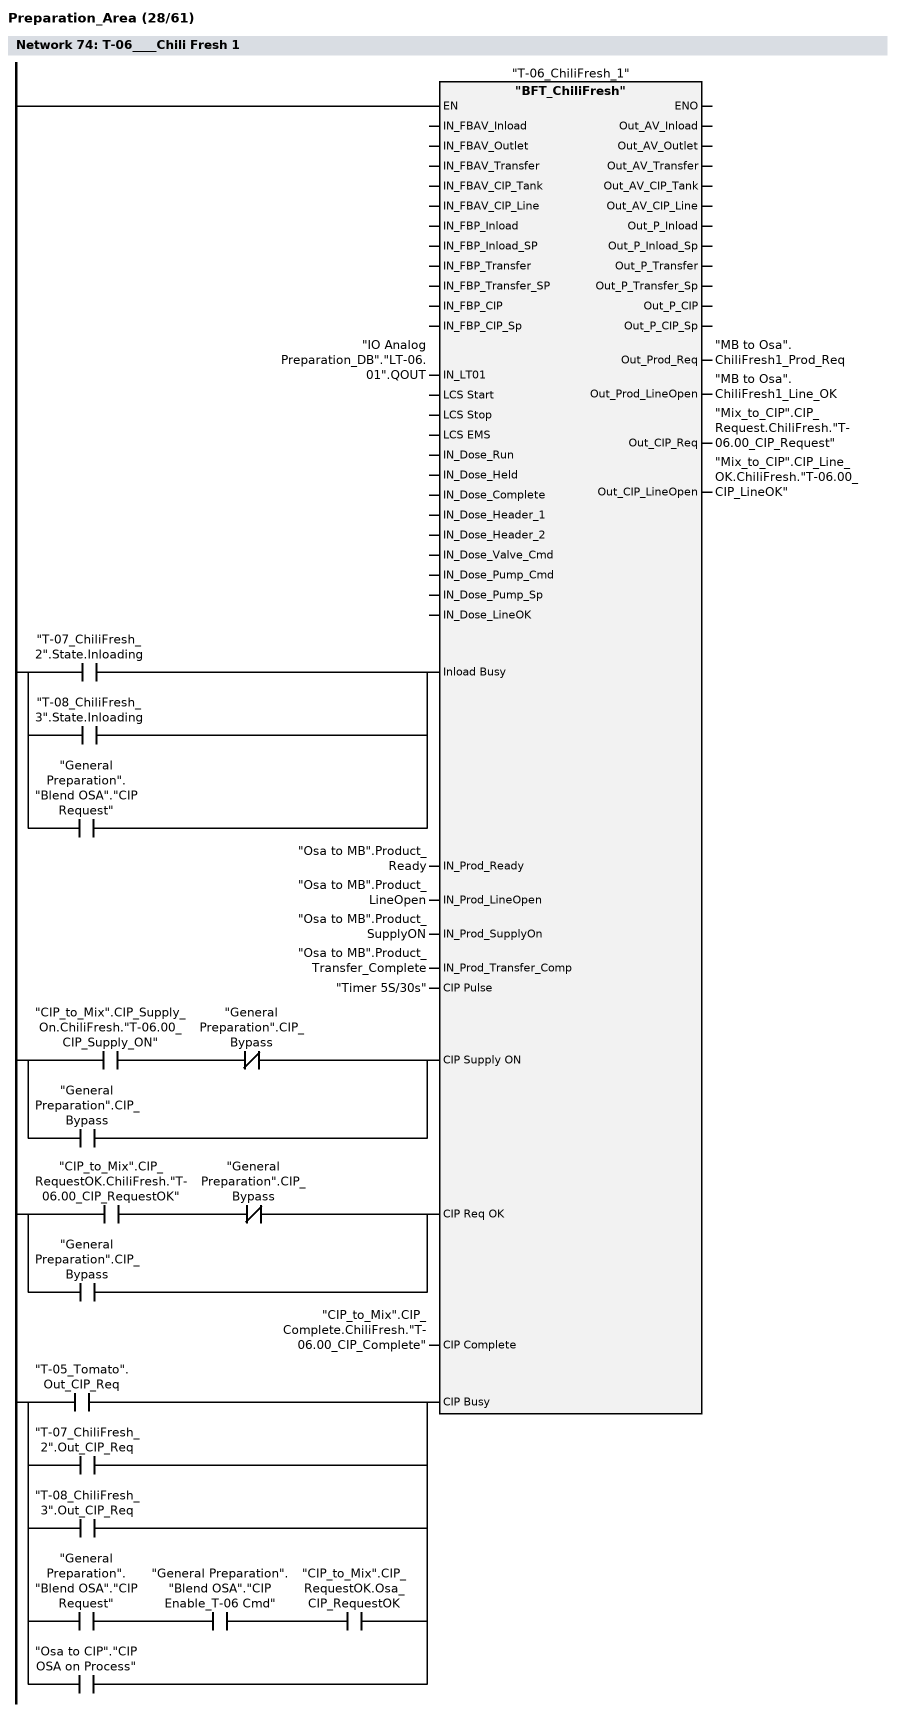
   RUNG wire#powerrail
      "T-06_ChiliFresh_1"("Inload Busy" := wire#w1, "CIP Supply ON" := wire#w2, "CIP Req OK" := wire#w3, "CIP Busy" := wire#w4, IN_FBAV_Inload :=, IN_FBAV_Outlet :=, IN_FBAV_Transfer :=, IN_FBAV_CIP_Tank :=, IN_FBAV_CIP_Line :=, IN_FBP_Inload :=, IN_FBP_Inload_SP :=, IN_FBP_Transfer :=, IN_FBP_Transfer_SP :=, IN_FBP_CIP :=, IN_FBP_CIP_Sp :=, IN_LT01 := "IO Analog Preparation_DB"."LT-06.01".QOUT, "LCS Start" :=, "LCS Stop" :=, "LCS EMS" :=, IN_Dose_Run :=, IN_Dose_Held :=, IN_Dose_Complete :=, IN_Dose_Header_1 :=, IN_Dose_Header_2 :=, IN_Dose_Valve_Cmd :=, IN_Dose_Pump_Cmd :=, IN_Dose_Pump_Sp :=, IN_Dose_LineOK :=, IN_Prod_Ready := "Osa to MB".Product_Ready, IN_Prod_LineOpen := "Osa to MB".Product_LineOpen, IN_Prod_SupplyOn := "Osa to MB".Product_SupplyON, IN_Prod_Transfer_Comp := "Osa to MB".Product_Transfer_Complete, "CIP Pulse" := "Timer 5S/30s", "CIP Complete" := "CIP_to_Mix".CIP_Complete.ChiliFresh."T-06.00_CIP_Complete", Out_AV_Inload =>, Out_AV_Outlet =>, Out_AV_Transfer =>, Out_AV_CIP_Tank =>, Out_AV_CIP_Line =>, Out_P_Inload =>, Out_P_Inload_Sp =>, Out_P_Transfer =>, Out_P_Transfer_Sp =>, Out_P_CIP =>, Out_P_CIP_Sp =>, Out_Prod_Req => "MB to Osa".ChiliFresh1_Prod_Req, Out_Prod_LineOpen => "MB to Osa".ChiliFresh1_Line_OK, Out_CIP_Req => "Mix_to_CIP".CIP_Request.ChiliFresh."T-06.00_CIP_Request", Out_CIP_LineOpen => "Mix_to_CIP".CIP_Line_OK.ChiliFresh."T-06.00_CIP_LineOK")
   END_RUNG
   RUNG wire#powerrail
      Contact( "T-07_ChiliFresh_2".State.Inloading )
   END_RUNG wire#w1
   RUNG wire#powerrail
      Contact( "T-08_ChiliFresh_3".State.Inloading )
   END_RUNG wire#w1
   RUNG wire#powerrail
      Contact( "General Preparation"."Blend OSA"."CIP Request" )
   END_RUNG wire#w1
   RUNG wire#powerrail
      Contact( "CIP_to_Mix".CIP_Supply_On.ChiliFresh."T-06.00_CIP_Supply_ON" )
      I_Contact( "General Preparation".CIP_Bypass )
   END_RUNG wire#w2
   RUNG wire#powerrail
      Contact( "General Preparation".CIP_Bypass )
   END_RUNG wire#w2
   RUNG wire#powerrail
      Contact( "CIP_to_Mix".CIP_RequestOK.ChiliFresh."T-06.00_CIP_RequestOK" )
      I_Contact( "General Preparation".CIP_Bypass )
   END_RUNG wire#w3
   RUNG wire#powerrail
      Contact( "General Preparation".CIP_Bypass )
   END_RUNG wire#w3
   RUNG wire#powerrail
      Contact( "T-05_Tomato".Out_CIP_Req )
   END_RUNG wire#w4
   RUNG wire#powerrail
      Contact( "T-07_ChiliFresh_2".Out_CIP_Req )
   END_RUNG wire#w4
   RUNG wire#powerrail
      Contact( "T-08_ChiliFresh_3".Out_CIP_Req )
   END_RUNG wire#w4
   RUNG wire#powerrail
      Contact( "General Preparation"."Blend OSA"."CIP Request" )
      Contact( "General Preparation"."Blend OSA"."CIP Enable_T-06 Cmd" )
      Contact( "CIP_to_Mix".CIP_RequestOK.Osa_CIP_RequestOK )
   END_RUNG wire#w4
   RUNG wire#powerrail
      Contact( "Osa to CIP"."CIP OSA on Process" )
   END_RUNG wire#w4
   // the same network as SCL:
   "T-06_ChiliFresh_1"(IN_LT01 := "IO Analog Preparation_DB"."LT-06.01".QOUT,   // "BFT_ChiliFresh"
                       "Inload Busy" := "T-07_ChiliFresh_2".State.Inloading OR "T-08_ChiliFresh_3".State.Inloading OR "General Preparation"."Blend OSA"."CIP Request",
                       IN_Prod_Ready := "Osa to MB".Product_Ready,
                       IN_Prod_LineOpen := "Osa to MB".Product_LineOpen,
                       IN_Prod_SupplyOn := "Osa to MB".Product_SupplyON,
                       IN_Prod_Transfer_Comp := "Osa to MB".Product_Transfer_Complete,
                       "CIP Pulse" := "Timer 5S/30s",
                       "CIP Supply ON" := ("CIP_to_Mix".CIP_Supply_On.ChiliFresh."T-06.00_CIP_Supply_ON" AND NOT "General Preparation".CIP_Bypass) OR "General Preparation".CIP_Bypass,
                       "CIP Req OK" := ("CIP_to_Mix".CIP_RequestOK.ChiliFresh."T-06.00_CIP_RequestOK" AND NOT "General Preparation".CIP_Bypass) OR "General Preparation".CIP_Bypass,
                       "CIP Complete" := "CIP_to_Mix".CIP_Complete.ChiliFresh."T-06.00_CIP_Complete",
                       "CIP Busy" := "T-05_Tomato".Out_CIP_Req OR "T-07_ChiliFresh_2".Out_CIP_Req OR "T-08_ChiliFresh_3".Out_CIP_Req OR ("General Preparation"."Blend OSA"."CIP Request" AND "General Preparation"."Blend OSA"."CIP Enable_T-06 Cmd" AND "CIP_to_Mix".CIP_RequestOK.Osa_CIP_RequestOK) OR "Osa to CIP"."CIP OSA on Process",
                       Out_Prod_Req => "MB to Osa".ChiliFresh1_Prod_Req,
                       Out_Prod_LineOpen => "MB to Osa".ChiliFresh1_Line_OK,
                       Out_CIP_Req => "Mix_to_CIP".CIP_Request.ChiliFresh."T-06.00_CIP_Request",
                       Out_CIP_LineOpen => "Mix_to_CIP".CIP_Line_OK.ChiliFresh."T-06.00_CIP_LineOK");
END_REGION

REGION Network 75: T-06.00 Valve Cmd
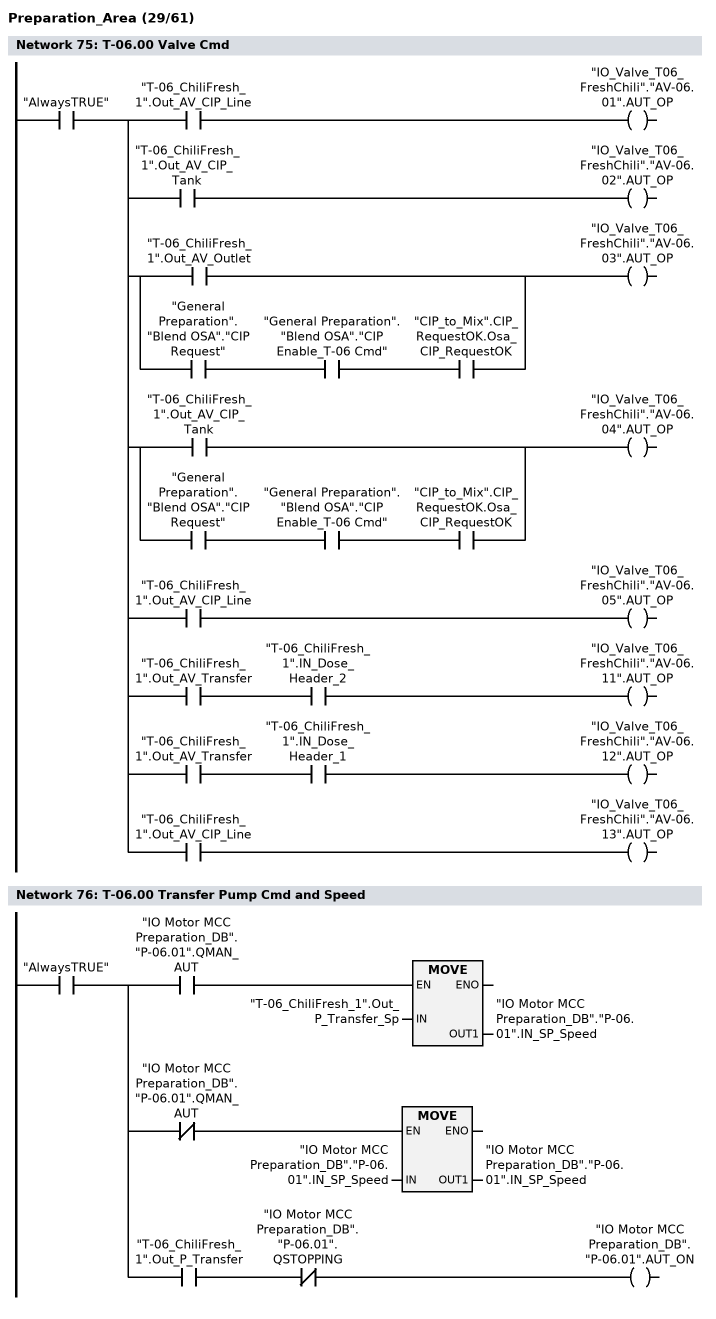
   RUNG wire#powerrail
      Contact( "AlwaysTRUE" )
      wire#w1
      Contact( "T-06_ChiliFresh_1".Out_AV_CIP_Line )
      Coil( "IO_Valve_T06_FreshChili"."AV-06.01".AUT_OP )
   END_RUNG
   RUNG wire#w1
      Contact( "T-06_ChiliFresh_1".Out_AV_CIP_Tank )
      Coil( "IO_Valve_T06_FreshChili"."AV-06.02".AUT_OP )
   END_RUNG
   RUNG wire#w1
      Contact( "T-06_ChiliFresh_1".Out_AV_Outlet )
      wire#w2
      Coil( "IO_Valve_T06_FreshChili"."AV-06.03".AUT_OP )
   END_RUNG
   RUNG wire#w1
      Contact( "General Preparation"."Blend OSA"."CIP Request" )
      Contact( "General Preparation"."Blend OSA"."CIP Enable_T-06 Cmd" )
      Contact( "CIP_to_Mix".CIP_RequestOK.Osa_CIP_RequestOK )
   END_RUNG wire#w2
   RUNG wire#w1
      Contact( "T-06_ChiliFresh_1".Out_AV_CIP_Tank )
      wire#w3
      Coil( "IO_Valve_T06_FreshChili"."AV-06.04".AUT_OP )
   END_RUNG
   RUNG wire#w1
      Contact( "General Preparation"."Blend OSA"."CIP Request" )
      Contact( "General Preparation"."Blend OSA"."CIP Enable_T-06 Cmd" )
      Contact( "CIP_to_Mix".CIP_RequestOK.Osa_CIP_RequestOK )
   END_RUNG wire#w3
   RUNG wire#w1
      Contact( "T-06_ChiliFresh_1".Out_AV_CIP_Line )
      Coil( "IO_Valve_T06_FreshChili"."AV-06.05".AUT_OP )
   END_RUNG
   RUNG wire#w1
      Contact( "T-06_ChiliFresh_1".Out_AV_Transfer )
      Contact( "T-06_ChiliFresh_1".IN_Dose_Header_2 )
      Coil( "IO_Valve_T06_FreshChili"."AV-06.11".AUT_OP )
   END_RUNG
   RUNG wire#w1
      Contact( "T-06_ChiliFresh_1".Out_AV_Transfer )
      Contact( "T-06_ChiliFresh_1".IN_Dose_Header_1 )
      Coil( "IO_Valve_T06_FreshChili"."AV-06.12".AUT_OP )
   END_RUNG
   RUNG wire#w1
      Contact( "T-06_ChiliFresh_1".Out_AV_CIP_Line )
      Coil( "IO_Valve_T06_FreshChili"."AV-06.13".AUT_OP )
   END_RUNG
   // the same network as SCL:
   "IO_Valve_T06_FreshChili"."AV-06.01".AUT_OP := "AlwaysTRUE" AND "T-06_ChiliFresh_1".Out_AV_CIP_Line;
   "IO_Valve_T06_FreshChili"."AV-06.02".AUT_OP := "AlwaysTRUE" AND "T-06_ChiliFresh_1".Out_AV_CIP_Tank;
   "IO_Valve_T06_FreshChili"."AV-06.03".AUT_OP := "AlwaysTRUE" AND ("T-06_ChiliFresh_1".Out_AV_Outlet OR ("General Preparation"."Blend OSA"."CIP Request" AND "General Preparation"."Blend OSA"."CIP Enable_T-06 Cmd" AND "CIP_to_Mix".CIP_RequestOK.Osa_CIP_RequestOK));
   "IO_Valve_T06_FreshChili"."AV-06.04".AUT_OP := "AlwaysTRUE" AND ("T-06_ChiliFresh_1".Out_AV_CIP_Tank OR ("General Preparation"."Blend OSA"."CIP Request" AND "General Preparation"."Blend OSA"."CIP Enable_T-06 Cmd" AND "CIP_to_Mix".CIP_RequestOK.Osa_CIP_RequestOK));
   "IO_Valve_T06_FreshChili"."AV-06.05".AUT_OP := "AlwaysTRUE" AND "T-06_ChiliFresh_1".Out_AV_CIP_Line;
   "IO_Valve_T06_FreshChili"."AV-06.11".AUT_OP := "AlwaysTRUE" AND "T-06_ChiliFresh_1".Out_AV_Transfer AND "T-06_ChiliFresh_1".IN_Dose_Header_2;
   "IO_Valve_T06_FreshChili"."AV-06.12".AUT_OP := "AlwaysTRUE" AND "T-06_ChiliFresh_1".Out_AV_Transfer AND "T-06_ChiliFresh_1".IN_Dose_Header_1;
   "IO_Valve_T06_FreshChili"."AV-06.13".AUT_OP := "AlwaysTRUE" AND "T-06_ChiliFresh_1".Out_AV_CIP_Line;
END_REGION

REGION Network 76: T-06.00 Transfer Pump Cmd and Speed
   RUNG wire#powerrail
      Contact( "AlwaysTRUE" )
      wire#w1
      Contact( "IO Motor MCC Preparation_DB"."P-06.01".QMAN_AUT )
      Move(in := "T-06_ChiliFresh_1".Out_P_Transfer_Sp, out1 => "IO Motor MCC Preparation_DB"."P-06.01".IN_SP_Speed)
   END_RUNG
   RUNG wire#w1
      I_Contact( "IO Motor MCC Preparation_DB"."P-06.01".QMAN_AUT )
      Move(in := "IO Motor MCC Preparation_DB"."P-06.01".IN_SP_Speed, out1 => "IO Motor MCC Preparation_DB"."P-06.01".IN_SP_Speed)
   END_RUNG
   RUNG wire#w1
      Contact( "T-06_ChiliFresh_1".Out_P_Transfer )
      I_Contact( "IO Motor MCC Preparation_DB"."P-06.01".QSTOPPING )
      Coil( "IO Motor MCC Preparation_DB"."P-06.01".AUT_ON )
   END_RUNG
   // the same network as SCL:
   IF "AlwaysTRUE" AND "IO Motor MCC Preparation_DB"."P-06.01".QMAN_AUT THEN
       "IO Motor MCC Preparation_DB"."P-06.01".IN_SP_Speed := "T-06_ChiliFresh_1".Out_P_Transfer_Sp;
   END_IF;
   IF "AlwaysTRUE" AND NOT "IO Motor MCC Preparation_DB"."P-06.01".QMAN_AUT THEN
       "IO Motor MCC Preparation_DB"."P-06.01".IN_SP_Speed := "IO Motor MCC Preparation_DB"."P-06.01".IN_SP_Speed;
   END_IF;
   "IO Motor MCC Preparation_DB"."P-06.01".AUT_ON := "AlwaysTRUE" AND "T-06_ChiliFresh_1".Out_P_Transfer AND NOT "IO Motor MCC Preparation_DB"."P-06.01".QSTOPPING;
END_REGION

REGION Network 77: T-06.00 Feedback Instrument
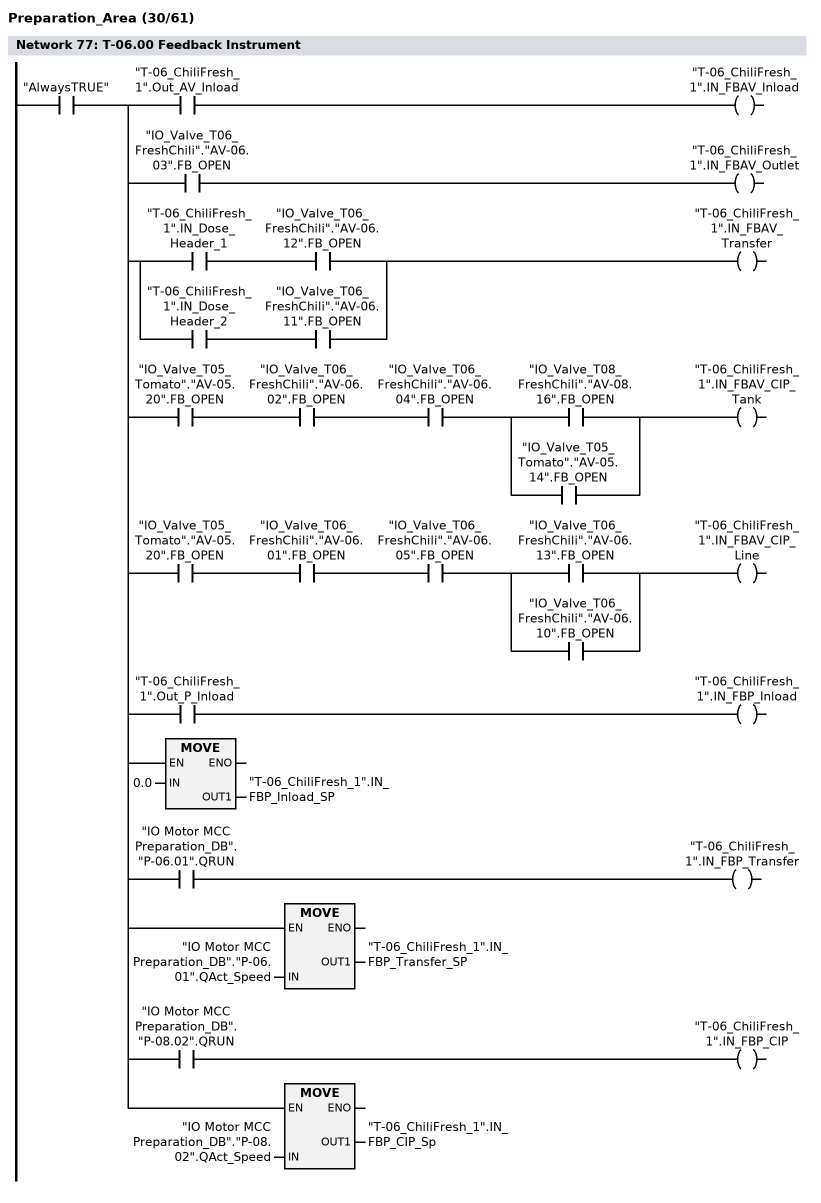
   RUNG wire#powerrail
      Contact( "AlwaysTRUE" )
      wire#w1
      Contact( "T-06_ChiliFresh_1".Out_AV_Inload )
      Coil( "T-06_ChiliFresh_1".IN_FBAV_Inload )
   END_RUNG
   RUNG wire#w1
      Contact( "IO_Valve_T06_FreshChili"."AV-06.03".FB_OPEN )
      Coil( "T-06_ChiliFresh_1".IN_FBAV_Outlet )
   END_RUNG
   RUNG wire#w1
      Contact( "T-06_ChiliFresh_1".IN_Dose_Header_1 )
      Contact( "IO_Valve_T06_FreshChili"."AV-06.12".FB_OPEN )
      wire#w2
      Coil( "T-06_ChiliFresh_1".IN_FBAV_Transfer )
   END_RUNG
   RUNG wire#w1
      Contact( "T-06_ChiliFresh_1".IN_Dose_Header_2 )
      Contact( "IO_Valve_T06_FreshChili"."AV-06.11".FB_OPEN )
   END_RUNG wire#w2
   RUNG wire#w1
      Contact( "IO_Valve_T05_Tomato"."AV-05.20".FB_OPEN )
      Contact( "IO_Valve_T06_FreshChili"."AV-06.02".FB_OPEN )
      Contact( "IO_Valve_T06_FreshChili"."AV-06.04".FB_OPEN )
      wire#w3
      Contact( "IO_Valve_T08_FreshChili"."AV-08.16".FB_OPEN )
      wire#w4
      Coil( "T-06_ChiliFresh_1".IN_FBAV_CIP_Tank )
   END_RUNG
   RUNG wire#w3
      Contact( "IO_Valve_T05_Tomato"."AV-05.14".FB_OPEN )
   END_RUNG wire#w4
   RUNG wire#w1
      Contact( "IO_Valve_T05_Tomato"."AV-05.20".FB_OPEN )
      Contact( "IO_Valve_T06_FreshChili"."AV-06.01".FB_OPEN )
      Contact( "IO_Valve_T06_FreshChili"."AV-06.05".FB_OPEN )
      wire#w5
      Contact( "IO_Valve_T06_FreshChili"."AV-06.13".FB_OPEN )
      wire#w6
      Coil( "T-06_ChiliFresh_1".IN_FBAV_CIP_Line )
   END_RUNG
   RUNG wire#w5
      Contact( "IO_Valve_T06_FreshChili"."AV-06.10".FB_OPEN )
   END_RUNG wire#w6
   RUNG wire#w1
      Contact( "T-06_ChiliFresh_1".Out_P_Inload )
      Coil( "T-06_ChiliFresh_1".IN_FBP_Inload )
   END_RUNG
   RUNG wire#w1
      Move(in := 0.0, out1 => "T-06_ChiliFresh_1".IN_FBP_Inload_SP)
   END_RUNG
   RUNG wire#w1
      Contact( "IO Motor MCC Preparation_DB"."P-06.01".QRUN )
      Coil( "T-06_ChiliFresh_1".IN_FBP_Transfer )
   END_RUNG
   RUNG wire#w1
      Move(in := "IO Motor MCC Preparation_DB"."P-06.01".QAct_Speed, out1 => "T-06_ChiliFresh_1".IN_FBP_Transfer_SP)
   END_RUNG
   RUNG wire#w1
      Contact( "IO Motor MCC Preparation_DB"."P-08.02".QRUN )
      Coil( "T-06_ChiliFresh_1".IN_FBP_CIP )
   END_RUNG
   RUNG wire#w1
      Move(in := "IO Motor MCC Preparation_DB"."P-08.02".QAct_Speed, out1 => "T-06_ChiliFresh_1".IN_FBP_CIP_Sp)
   END_RUNG
   // the same network as SCL:
   "T-06_ChiliFresh_1".IN_FBAV_Inload := "AlwaysTRUE" AND "T-06_ChiliFresh_1".Out_AV_Inload;
   "T-06_ChiliFresh_1".IN_FBAV_Outlet := "AlwaysTRUE" AND "IO_Valve_T06_FreshChili"."AV-06.03".FB_OPEN;
   "T-06_ChiliFresh_1".IN_FBAV_Transfer := "AlwaysTRUE" AND (("T-06_ChiliFresh_1".IN_Dose_Header_1 AND "IO_Valve_T06_FreshChili"."AV-06.12".FB_OPEN) OR ("T-06_ChiliFresh_1".IN_Dose_Header_2 AND "IO_Valve_T06_FreshChili"."AV-06.11".FB_OPEN));
   "T-06_ChiliFresh_1".IN_FBAV_CIP_Tank := "AlwaysTRUE" AND "IO_Valve_T05_Tomato"."AV-05.20".FB_OPEN AND "IO_Valve_T06_FreshChili"."AV-06.02".FB_OPEN AND "IO_Valve_T06_FreshChili"."AV-06.04".FB_OPEN AND ("IO_Valve_T08_FreshChili"."AV-08.16".FB_OPEN OR "IO_Valve_T05_Tomato"."AV-05.14".FB_OPEN);
   "T-06_ChiliFresh_1".IN_FBAV_CIP_Line := "AlwaysTRUE" AND "IO_Valve_T05_Tomato"."AV-05.20".FB_OPEN AND "IO_Valve_T06_FreshChili"."AV-06.01".FB_OPEN AND "IO_Valve_T06_FreshChili"."AV-06.05".FB_OPEN AND ("IO_Valve_T06_FreshChili"."AV-06.13".FB_OPEN OR "IO_Valve_T06_FreshChili"."AV-06.10".FB_OPEN);
   "T-06_ChiliFresh_1".IN_FBP_Inload := "AlwaysTRUE" AND "T-06_ChiliFresh_1".Out_P_Inload;
   IF "AlwaysTRUE" THEN "T-06_ChiliFresh_1".IN_FBP_Inload_SP := 0.0; END_IF;
   "T-06_ChiliFresh_1".IN_FBP_Transfer := "AlwaysTRUE" AND "IO Motor MCC Preparation_DB"."P-06.01".QRUN;
   IF "AlwaysTRUE" THEN
       "T-06_ChiliFresh_1".IN_FBP_Transfer_SP := "IO Motor MCC Preparation_DB"."P-06.01".QAct_Speed;
   END_IF;
   "T-06_ChiliFresh_1".IN_FBP_CIP := "AlwaysTRUE" AND "IO Motor MCC Preparation_DB"."P-08.02".QRUN;
   IF "AlwaysTRUE" THEN
       "T-06_ChiliFresh_1".IN_FBP_CIP_Sp := "IO Motor MCC Preparation_DB"."P-08.02".QAct_Speed;
   END_IF;
END_REGION

REGION Network 78: T-06.00 Comm to Blend
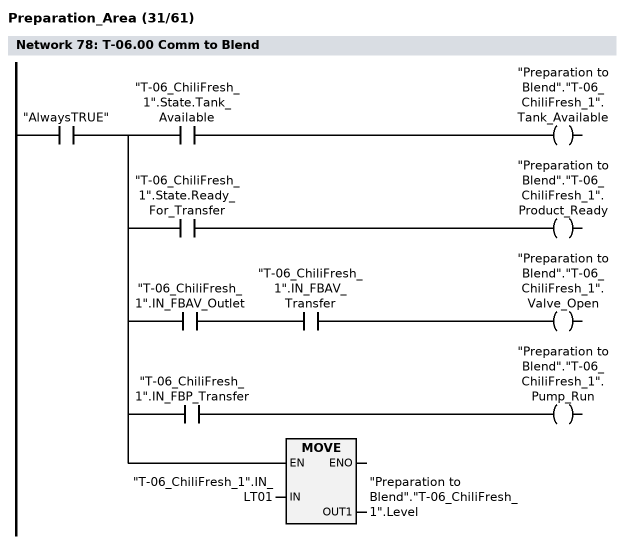
   RUNG wire#powerrail
      Contact( "AlwaysTRUE" )
      wire#w1
      Contact( "T-06_ChiliFresh_1".State.Tank_Available )
      Coil( "Preparation to Blend"."T-06_ChiliFresh_1".Tank_Available )
   END_RUNG
   RUNG wire#w1
      Contact( "T-06_ChiliFresh_1".State.Ready_For_Transfer )
      Coil( "Preparation to Blend"."T-06_ChiliFresh_1".Product_Ready )
   END_RUNG
   RUNG wire#w1
      Contact( "T-06_ChiliFresh_1".IN_FBAV_Outlet )
      Contact( "T-06_ChiliFresh_1".IN_FBAV_Transfer )
      Coil( "Preparation to Blend"."T-06_ChiliFresh_1".Valve_Open )
   END_RUNG
   RUNG wire#w1
      Contact( "T-06_ChiliFresh_1".IN_FBP_Transfer )
      Coil( "Preparation to Blend"."T-06_ChiliFresh_1".Pump_Run )
   END_RUNG
   RUNG wire#w1
      Move(in := "T-06_ChiliFresh_1".IN_LT01, out1 => "Preparation to Blend"."T-06_ChiliFresh_1".Level)
   END_RUNG
   // the same network as SCL:
   "Preparation to Blend"."T-06_ChiliFresh_1".Tank_Available := "AlwaysTRUE" AND "T-06_ChiliFresh_1".State.Tank_Available;
   "Preparation to Blend"."T-06_ChiliFresh_1".Product_Ready := "AlwaysTRUE" AND "T-06_ChiliFresh_1".State.Ready_For_Transfer;
   "Preparation to Blend"."T-06_ChiliFresh_1".Valve_Open := "AlwaysTRUE" AND "T-06_ChiliFresh_1".IN_FBAV_Outlet AND "T-06_ChiliFresh_1".IN_FBAV_Transfer;
   "Preparation to Blend"."T-06_ChiliFresh_1".Pump_Run := "AlwaysTRUE" AND "T-06_ChiliFresh_1".IN_FBP_Transfer;
   IF "AlwaysTRUE" THEN
       "Preparation to Blend"."T-06_ChiliFresh_1".Level := "T-06_ChiliFresh_1".IN_LT01;
   END_IF;
END_REGION

NETWORK
TITLE = T-07.00 DOSE ON OFF
      O     "Blend to Preparation"."T-20".Raw_Material.ChiliFresh_2.DoseRun;
      O     "Blend to Preparation"."T-21".Raw_Material.ChiliFresh_2.DoseRun;
      O     "Blend to Preparation"."T-30".Raw_Material.ChiliFresh_2.DoseRun;
      O     "Blend to Preparation"."T-31".Raw_Material.ChiliFresh_2.DoseRun;
      O     "Blend to Preparation"."T-40".Raw_Material.ChiliFresh_2.DoseRun;
      O     "Blend to Preparation"."T-41".Raw_Material.ChiliFresh_2.DoseRun;
      =     "T-07_ChiliFresh_2".IN_Dose_Run;

NETWORK
TITLE = T-07.00 DOSE PAUSE
      O     "Blend to Preparation"."T-20".Raw_Material.ChiliFresh_2.DoseHeld;
      O     "Blend to Preparation"."T-21".Raw_Material.ChiliFresh_2.DoseHeld;
      O     "Blend to Preparation"."T-30".Raw_Material.ChiliFresh_2.DoseHeld;
      O     "Blend to Preparation"."T-31".Raw_Material.ChiliFresh_2.DoseHeld;
      O     "Blend to Preparation"."T-40".Raw_Material.ChiliFresh_2.DoseHeld;
      O     "Blend to Preparation"."T-41".Raw_Material.ChiliFresh_2.DoseHeld;
      =     "T-07_ChiliFresh_2".IN_Dose_Held;

NETWORK
TITLE = T-07.00 DOSE VALVE CMD
      O(;
      A     "Blend to Preparation"."T-20".Raw_Material.ChiliFresh_2.DoseRun;
      A     "Blend to Preparation"."T-20".Raw_Material.ChiliFresh_2.ValveCMD;
      );
      O(;
      A     "Blend to Preparation"."T-21".Raw_Material.ChiliFresh_2.DoseRun;
      A     "Blend to Preparation"."T-21".Raw_Material.ChiliFresh_2.ValveCMD;
      );
      O(;
      A     "Blend to Preparation"."T-30".Raw_Material.ChiliFresh_2.DoseRun;
      A     "Blend to Preparation"."T-30".Raw_Material.ChiliFresh_2.ValveCMD;
      );
      O(;
      A     "Blend to Preparation"."T-31".Raw_Material.ChiliFresh_2.DoseRun;
      A     "Blend to Preparation"."T-31".Raw_Material.ChiliFresh_2.ValveCMD;
      );
      O(;
      A     "Blend to Preparation"."T-40".Raw_Material.ChiliFresh_2.DoseRun;
      A     "Blend to Preparation"."T-40".Raw_Material.ChiliFresh_2.ValveCMD;
      );
      O(;
      A     "Blend to Preparation"."T-41".Raw_Material.ChiliFresh_2.DoseRun;
      A     "Blend to Preparation"."T-41".Raw_Material.ChiliFresh_2.ValveCMD;
      );
      =     "T-07_ChiliFresh_2".IN_Dose_Valve_Cmd;



NETWORK
TITLE = T-07.00 DOSE Pump CMD
      O(;
      A     "Blend to Preparation"."T-20".Raw_Material.ChiliFresh_2.DoseRun;
      A     "Blend to Preparation"."T-20".Raw_Material.ChiliFresh_2.PumpCMD;
      );
      O(;
      A     "Blend to Preparation"."T-21".Raw_Material.ChiliFresh_2.DoseRun;
      A     "Blend to Preparation"."T-21".Raw_Material.ChiliFresh_2.PumpCMD;
      );
      O(;
      A     "Blend to Preparation"."T-30".Raw_Material.ChiliFresh_2.DoseRun;
      A     "Blend to Preparation"."T-30".Raw_Material.ChiliFresh_2.PumpCMD;
      );
      O(;
      A     "Blend to Preparation"."T-31".Raw_Material.ChiliFresh_2.DoseRun;
      A     "Blend to Preparation"."T-31".Raw_Material.ChiliFresh_2.PumpCMD;
      );
      O(;
      A     "Blend to Preparation"."T-40".Raw_Material.ChiliFresh_2.DoseRun;
      A     "Blend to Preparation"."T-40".Raw_Material.ChiliFresh_2.PumpCMD;
      );
      O(;
      A     "Blend to Preparation"."T-41".Raw_Material.ChiliFresh_2.DoseRun;
      A     "Blend to Preparation"."T-41".Raw_Material.ChiliFresh_2.PumpCMD;
      );
      =     "T-07_ChiliFresh_2".IN_Dose_Pump_Cmd;



NETWORK
TITLE = T-07.00 DOSE PUMP SPEED
// Checking
      O     "Blend to Preparation"."T-20".Raw_Material.ChiliFresh_2.DoseRun;
      JC    SP_07_FROM_20;
      O     "Blend to Preparation"."T-21".Raw_Material.ChiliFresh_2.DoseRun;
      JC    SP_07_FROM_21;
      O     "Blend to Preparation"."T-30".Raw_Material.ChiliFresh_2.DoseRun;
      JC    SP_07_FROM_30;
      O     "Blend to Preparation"."T-31".Raw_Material.ChiliFresh_2.DoseRun;
      JC    SP_07_FROM_31;
      O     "Blend to Preparation"."T-40".Raw_Material.ChiliFresh_2.DoseRun;
      JC    SP_07_FROM_40;
      O     "Blend to Preparation"."T-41".Raw_Material.ChiliFresh_2.DoseRun;
      JC    SP_07_FROM_41;
//Jump to end if Blend not Dosing
      JC    SP_07_SELF;
//Load Set Point
SP_07_FROM_20:L     "Blend to Preparation".Recipe."T-20".ChiliFresh_2.SP_PumpSpeed;
      T     "T-07_ChiliFresh_2".IN_Dose_Pump_Sp;
      JC    SP_07_SELF;
SP_07_FROM_21:L     "Blend to Preparation".Recipe."T-21".ChiliFresh_2.SP_PumpSpeed;
      T     "T-07_ChiliFresh_2".IN_Dose_Pump_Sp;
      JC    SP_07_SELF;
SP_07_FROM_30:L     "Blend to Preparation".Recipe."T-30".ChiliFresh_2.SP_PumpSpeed;
      T     "T-07_ChiliFresh_2".IN_Dose_Pump_Sp;
      JC    SP_07_SELF;
SP_07_FROM_31:L     "Blend to Preparation".Recipe."T-31".ChiliFresh_2.SP_PumpSpeed;
      T     "T-07_ChiliFresh_2".IN_Dose_Pump_Sp;
      JC    SP_07_SELF;
SP_07_FROM_40:L     "Blend to Preparation".Recipe."T-40".ChiliFresh_2.SP_PumpSpeed;
      T     "T-07_ChiliFresh_2".IN_Dose_Pump_Sp;
      JC    SP_07_SELF;
SP_07_FROM_41:L     "Blend to Preparation".Recipe."T-41".ChiliFresh_2.SP_PumpSpeed;
      T     "T-07_ChiliFresh_2".IN_Dose_Pump_Sp;
      JC    SP_07_SELF;
// END
SP_07_SELF:L     "T-07_ChiliFresh_2".IN_Dose_Pump_Sp;
      T     "T-07_ChiliFresh_2".IN_Dose_Pump_Sp;


NETWORK
TITLE = T-07.00 Header Req
// HEADER 1 Req
      O     "Blend to Preparation"."T-20".Raw_Material.ChiliFresh_2.Header1_Req;
      O     "Blend to Preparation"."T-21".Raw_Material.ChiliFresh_2.Header1_Req;
      O     "Blend to Preparation"."T-30".Raw_Material.ChiliFresh_2.Header1_Req;
      O     "Blend to Preparation"."T-31".Raw_Material.ChiliFresh_2.Header1_Req;
      O     "Blend to Preparation"."T-40".Raw_Material.ChiliFresh_2.Header1_Req;
      O     "Blend to Preparation"."T-41".Raw_Material.ChiliFresh_2.Header1_Req;
      =     "T-07_ChiliFresh_2".IN_Dose_Header_1;

// HEADER 2 Req
      O     "Blend to Preparation"."T-20".Raw_Material.ChiliFresh_2.Header2_Req;
      O     "Blend to Preparation"."T-21".Raw_Material.ChiliFresh_2.Header2_Req;
      O     "Blend to Preparation"."T-30".Raw_Material.ChiliFresh_2.Header2_Req;
      O     "Blend to Preparation"."T-31".Raw_Material.ChiliFresh_2.Header2_Req;
      O     "Blend to Preparation"."T-40".Raw_Material.ChiliFresh_2.Header2_Req;
      O     "Blend to Preparation"."T-41".Raw_Material.ChiliFresh_2.Header2_Req;
      =     "T-07_ChiliFresh_2".IN_Dose_Header_2;


REGION Network 87: T-07.00 LineTransferOK
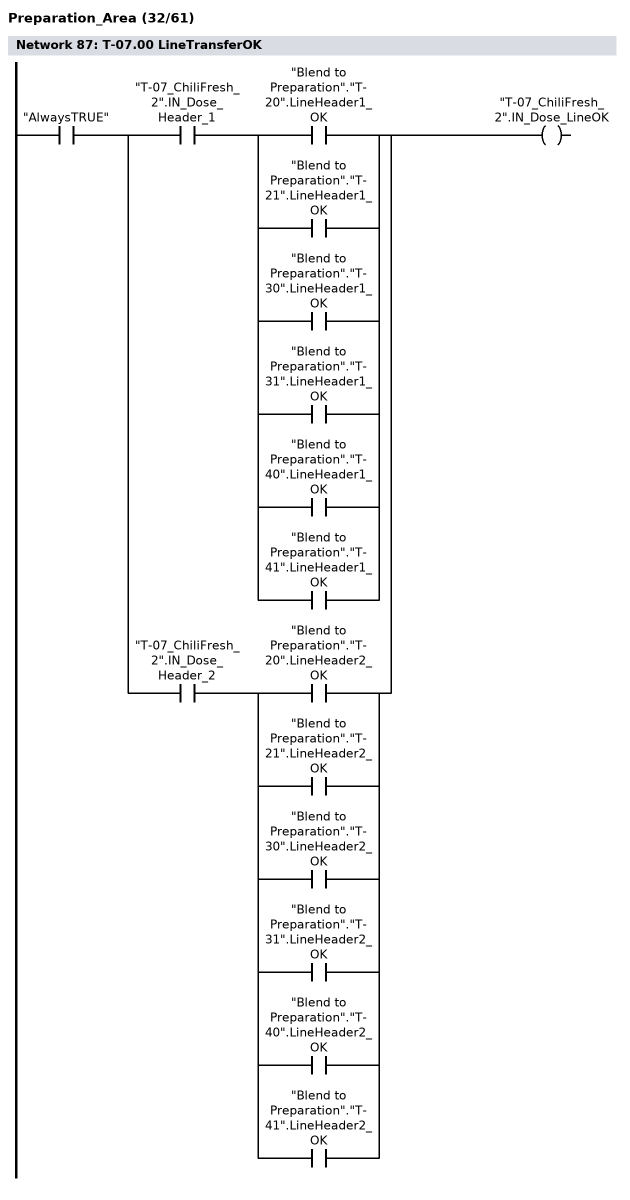
   RUNG wire#powerrail
      Contact( "AlwaysTRUE" )
      wire#w1
      Contact( "T-07_ChiliFresh_2".IN_Dose_Header_1 )
      wire#w2
      Contact( "Blend to Preparation"."T-20".LineHeader1_OK )
      wire#w3
      Coil( "T-07_ChiliFresh_2".IN_Dose_LineOK )
   END_RUNG
   RUNG wire#w2
      Contact( "Blend to Preparation"."T-21".LineHeader1_OK )
   END_RUNG wire#w3
   RUNG wire#w2
      Contact( "Blend to Preparation"."T-30".LineHeader1_OK )
   END_RUNG wire#w3
   RUNG wire#w2
      Contact( "Blend to Preparation"."T-31".LineHeader1_OK )
   END_RUNG wire#w3
   RUNG wire#w2
      Contact( "Blend to Preparation"."T-40".LineHeader1_OK )
   END_RUNG wire#w3
   RUNG wire#w2
      Contact( "Blend to Preparation"."T-41".LineHeader1_OK )
   END_RUNG wire#w3
   RUNG wire#w1
      Contact( "T-07_ChiliFresh_2".IN_Dose_Header_2 )
      wire#w4
      Contact( "Blend to Preparation"."T-20".LineHeader2_OK )
   END_RUNG wire#w3
   RUNG wire#w4
      Contact( "Blend to Preparation"."T-21".LineHeader2_OK )
   END_RUNG wire#w3
   RUNG wire#w4
      Contact( "Blend to Preparation"."T-30".LineHeader2_OK )
   END_RUNG wire#w3
   RUNG wire#w4
      Contact( "Blend to Preparation"."T-31".LineHeader2_OK )
   END_RUNG wire#w3
   RUNG wire#w4
      Contact( "Blend to Preparation"."T-40".LineHeader2_OK )
   END_RUNG wire#w3
   RUNG wire#w4
      Contact( "Blend to Preparation"."T-41".LineHeader2_OK )
   END_RUNG wire#w3
   // the same network as SCL:
   "T-07_ChiliFresh_2".IN_Dose_LineOK := "AlwaysTRUE" AND (("T-07_ChiliFresh_2".IN_Dose_Header_1 AND ("Blend to Preparation"."T-20".LineHeader1_OK OR "Blend to Preparation"."T-21".LineHeader1_OK OR "Blend to Preparation"."T-30".LineHeader1_OK OR "Blend to Preparation"."T-31".LineHeader1_OK OR "Blend to Preparation"."T-40".LineHeader1_OK OR "Blend to Preparation"."T-41".LineHeader1_OK)) OR ("T-07_ChiliFresh_2".IN_Dose_Header_2 AND ("Blend to Preparation"."T-20".LineHeader2_OK OR "Blend to Preparation"."T-21".LineHeader2_OK OR "Blend to Preparation"."T-30".LineHeader2_OK OR "Blend to Preparation"."T-31".LineHeader2_OK OR "Blend to Preparation"."T-40".LineHeader2_OK OR "Blend to Preparation"."T-41".LineHeader2_OK)));
END_REGION

REGION Network 88: T-07____Chili Fresh 2
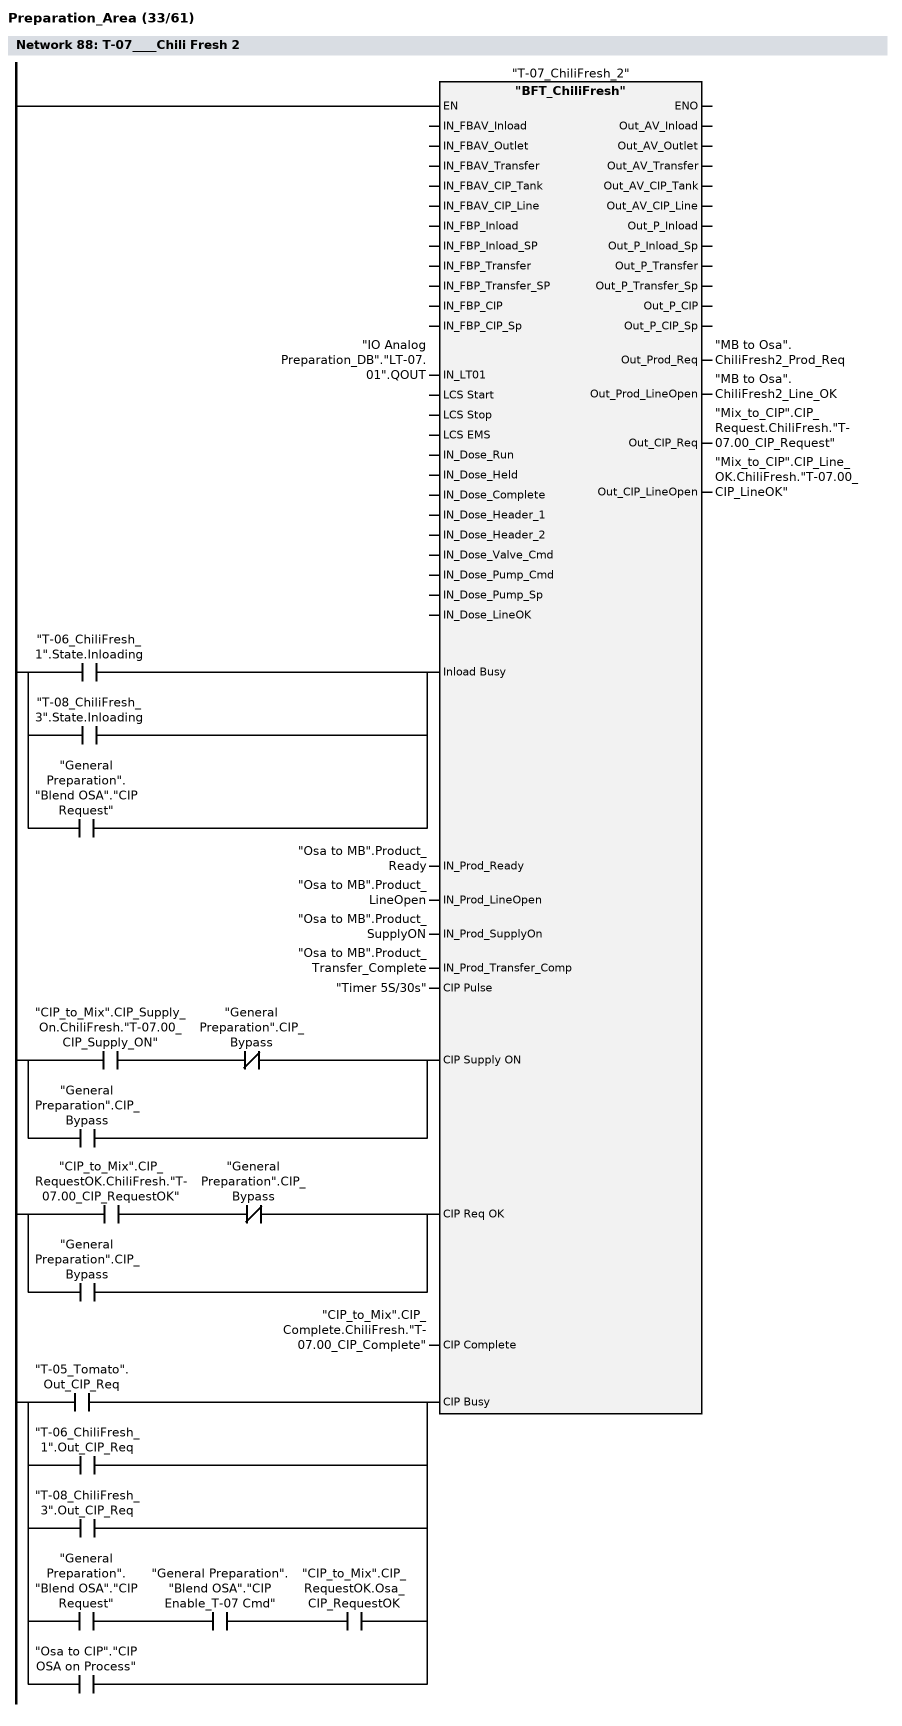
   RUNG wire#powerrail
      "T-07_ChiliFresh_2"("Inload Busy" := wire#w1, "CIP Supply ON" := wire#w2, "CIP Req OK" := wire#w3, "CIP Busy" := wire#w4, IN_FBAV_Inload :=, IN_FBAV_Outlet :=, IN_FBAV_Transfer :=, IN_FBAV_CIP_Tank :=, IN_FBAV_CIP_Line :=, IN_FBP_Inload :=, IN_FBP_Inload_SP :=, IN_FBP_Transfer :=, IN_FBP_Transfer_SP :=, IN_FBP_CIP :=, IN_FBP_CIP_Sp :=, IN_LT01 := "IO Analog Preparation_DB"."LT-07.01".QOUT, "LCS Start" :=, "LCS Stop" :=, "LCS EMS" :=, IN_Dose_Run :=, IN_Dose_Held :=, IN_Dose_Complete :=, IN_Dose_Header_1 :=, IN_Dose_Header_2 :=, IN_Dose_Valve_Cmd :=, IN_Dose_Pump_Cmd :=, IN_Dose_Pump_Sp :=, IN_Dose_LineOK :=, IN_Prod_Ready := "Osa to MB".Product_Ready, IN_Prod_LineOpen := "Osa to MB".Product_LineOpen, IN_Prod_SupplyOn := "Osa to MB".Product_SupplyON, IN_Prod_Transfer_Comp := "Osa to MB".Product_Transfer_Complete, "CIP Pulse" := "Timer 5S/30s", "CIP Complete" := "CIP_to_Mix".CIP_Complete.ChiliFresh."T-07.00_CIP_Complete", Out_AV_Inload =>, Out_AV_Outlet =>, Out_AV_Transfer =>, Out_AV_CIP_Tank =>, Out_AV_CIP_Line =>, Out_P_Inload =>, Out_P_Inload_Sp =>, Out_P_Transfer =>, Out_P_Transfer_Sp =>, Out_P_CIP =>, Out_P_CIP_Sp =>, Out_Prod_Req => "MB to Osa".ChiliFresh2_Prod_Req, Out_Prod_LineOpen => "MB to Osa".ChiliFresh2_Line_OK, Out_CIP_Req => "Mix_to_CIP".CIP_Request.ChiliFresh."T-07.00_CIP_Request", Out_CIP_LineOpen => "Mix_to_CIP".CIP_Line_OK.ChiliFresh."T-07.00_CIP_LineOK")
   END_RUNG
   RUNG wire#powerrail
      Contact( "T-06_ChiliFresh_1".State.Inloading )
   END_RUNG wire#w1
   RUNG wire#powerrail
      Contact( "T-08_ChiliFresh_3".State.Inloading )
   END_RUNG wire#w1
   RUNG wire#powerrail
      Contact( "General Preparation"."Blend OSA"."CIP Request" )
   END_RUNG wire#w1
   RUNG wire#powerrail
      Contact( "CIP_to_Mix".CIP_Supply_On.ChiliFresh."T-07.00_CIP_Supply_ON" )
      I_Contact( "General Preparation".CIP_Bypass )
   END_RUNG wire#w2
   RUNG wire#powerrail
      Contact( "General Preparation".CIP_Bypass )
   END_RUNG wire#w2
   RUNG wire#powerrail
      Contact( "CIP_to_Mix".CIP_RequestOK.ChiliFresh."T-07.00_CIP_RequestOK" )
      I_Contact( "General Preparation".CIP_Bypass )
   END_RUNG wire#w3
   RUNG wire#powerrail
      Contact( "General Preparation".CIP_Bypass )
   END_RUNG wire#w3
   RUNG wire#powerrail
      Contact( "T-05_Tomato".Out_CIP_Req )
   END_RUNG wire#w4
   RUNG wire#powerrail
      Contact( "T-06_ChiliFresh_1".Out_CIP_Req )
   END_RUNG wire#w4
   RUNG wire#powerrail
      Contact( "T-08_ChiliFresh_3".Out_CIP_Req )
   END_RUNG wire#w4
   RUNG wire#powerrail
      Contact( "General Preparation"."Blend OSA"."CIP Request" )
      Contact( "General Preparation"."Blend OSA"."CIP Enable_T-07 Cmd" )
      Contact( "CIP_to_Mix".CIP_RequestOK.Osa_CIP_RequestOK )
   END_RUNG wire#w4
   RUNG wire#powerrail
      Contact( "Osa to CIP"."CIP OSA on Process" )
   END_RUNG wire#w4
   // the same network as SCL:
   "T-07_ChiliFresh_2"(IN_LT01 := "IO Analog Preparation_DB"."LT-07.01".QOUT,   // "BFT_ChiliFresh"
                       "Inload Busy" := "T-06_ChiliFresh_1".State.Inloading OR "T-08_ChiliFresh_3".State.Inloading OR "General Preparation"."Blend OSA"."CIP Request",
                       IN_Prod_Ready := "Osa to MB".Product_Ready,
                       IN_Prod_LineOpen := "Osa to MB".Product_LineOpen,
                       IN_Prod_SupplyOn := "Osa to MB".Product_SupplyON,
                       IN_Prod_Transfer_Comp := "Osa to MB".Product_Transfer_Complete,
                       "CIP Pulse" := "Timer 5S/30s",
                       "CIP Supply ON" := ("CIP_to_Mix".CIP_Supply_On.ChiliFresh."T-07.00_CIP_Supply_ON" AND NOT "General Preparation".CIP_Bypass) OR "General Preparation".CIP_Bypass,
                       "CIP Req OK" := ("CIP_to_Mix".CIP_RequestOK.ChiliFresh."T-07.00_CIP_RequestOK" AND NOT "General Preparation".CIP_Bypass) OR "General Preparation".CIP_Bypass,
                       "CIP Complete" := "CIP_to_Mix".CIP_Complete.ChiliFresh."T-07.00_CIP_Complete",
                       "CIP Busy" := "T-05_Tomato".Out_CIP_Req OR "T-06_ChiliFresh_1".Out_CIP_Req OR "T-08_ChiliFresh_3".Out_CIP_Req OR ("General Preparation"."Blend OSA"."CIP Request" AND "General Preparation"."Blend OSA"."CIP Enable_T-07 Cmd" AND "CIP_to_Mix".CIP_RequestOK.Osa_CIP_RequestOK) OR "Osa to CIP"."CIP OSA on Process",
                       Out_Prod_Req => "MB to Osa".ChiliFresh2_Prod_Req,
                       Out_Prod_LineOpen => "MB to Osa".ChiliFresh2_Line_OK,
                       Out_CIP_Req => "Mix_to_CIP".CIP_Request.ChiliFresh."T-07.00_CIP_Request",
                       Out_CIP_LineOpen => "Mix_to_CIP".CIP_Line_OK.ChiliFresh."T-07.00_CIP_LineOK");
END_REGION

